  PRC_SendeKanalOeffnen()
  IF N_PRC_Err1 <> N_PRC_MsgOff THEN
    RETURN(N_PRC_Err1)
  ENDIF
  O_PRC_Data2 = 0
  O_PRC_Data1 = N_PRC_ID
  IF NOT PRC_DatenSenden() THEN
    RETURN(N_PRC_Err1)
  ENDIF
  PRC_SendeKanalSchliessen()
  IF NOT PRC_DatenEmpfangen() THEN
    RETURN(N_PRC_Err1)
  ENDIF
  PRC_EmpfKanalSchliessen()               ; PRC_EmpfKanalSchliessen
  PRC_EmpfDatenAuswerten()                ; PRC_EmpfDatenAuswerten
  IF N_PRC_IDAck <> N_PRC_ID THEN
    N_PRC_Err1   = N_PRC_MsgOff + 43      ; falsche RETURNID
    B_PRC_MsgFlg = TRUE
    RETURN(N_PRC_Err1)
  ENDIF
  SWITCH N_PRC_KennAck
    CASE 0
      N_PRC_Err1   = N_PRC_MsgOff         ; Perceptron bereit
    CASE 5
      N_PRC_Err1   = N_PRC_MsgOff + 7     ; Perceptron von diesem Roboter bereits gestartet
    CASE 12
      N_PRC_Err1   = N_PRC_MsgOff + 6     ; Perceptron offline
    CASE 23
      N_PRC_Err1   = N_PRC_MsgOff + 23    ; Kalibriermodus
    CASE 24
      N_PRC_Err1   = N_PRC_MsgOff + 24    ; Teachmodus
    CASE 29
      N_PRC_Err1   = N_PRC_MsgOff + 29    ; BaseFinder
    CASE 30
      N_PRC_Err1   = N_PRC_MsgOff + 30    ; ToolFinder
    CASE 255
      N_PRC_Err1   = N_PRC_MsgOff + 8     ; allg. Fehler
    DEFAULT
      N_PRC_Err1   = N_PRC_MsgOff + 9     ; Fehler nicht spezifiziert
  ENDSWITCH
  RETURN(N_PRC_Err1)
ENDFCT
;
  ;ENDFOLD (Get Status)
;
  ;FOLD Punkt Messung
;
DEF PRC_PunktMessung(nPktNr:IN,nFrame:IN,nTool:IN)
INT nPktNr
INT nFrame
INT nTool
INT nMPTimerStart
INT nComTimerStart
  N_PRC_Err1   = 200
  B_PRC_MsgFlg = FALSE
  IF (NOT I_PRC_Zyklus) AND (NOT I_PRC_PgmMod) THEN
    B_PRC_MsgFlg = TRUE
    N_PRC_Err1   = 224   ; Messung nicht gestartet
    RETURN
  ENDIF
  O_PRC_PktNr = nPktNr
  O_PRC_Pkt   = TRUE
  nMPTimerStart = $Rob_Timer
  wait for (I_PRC_PktAck OR I_PRC_PosInf OR ((($Rob_Timer - nMPTimerStart) > N_PRC_TmMP) AND NOT I_PRC_PgmMod))
  IF (($Rob_Timer - nMPTimerStart) > N_PRC_TmMP) AND NOT I_PRC_PgmMod THEN
    N_PRC_Err1   = 225   ; Timeout beim warten auf Messungende
    B_PRC_MsgFlg = TRUE
    O_PRC_PktNr  = 0
    O_PRC_Pkt    = FALSE
    RETURN
  ENDIF
  IF I_PRC_Fehler THEN   ; Perceptron Fehler bei PRC_PunktMessung
    B_PRC_MsgFlg = TRUE
    SWITCH I_PRC_FehlNr
      CASE 1
        N_PRC_Err1 = 223   ; PositionsID ungueltig
      CASE 5
        N_PRC_Err1 = 224   ; Messytstem nicht gestartet
      CASE 18
        N_PRC_Err1 = 213   ; Allgemeiner Fehler
      CASE 19
        N_PRC_Err1 = 227   ; Falsche Punktreihenfolge
CASE 512
        N_PRC_Err1 = 213   ; Allgemeiner Fehler
        IF B_PRC_ISTOOL == TRUE THEN
          N_PRC_Err1   = 228   ; Nur im ToolFinder-Modus (Messfehler)
          B_PRC_MsgFlg = FALSE
        ENDIF
        IF B_PRC_ISBASE == TRUE THEN
          N_PRC_Err1   = 229   ; Nur im BaseFinder-Modus (Messfehler)
          B_PRC_MsgFlg = FALSE
        ENDIF
      DEFAULT
    ENDSWITCH
    O_PRC_PktNr = 0
    O_PRC_Pkt   = FALSE
    RETURN
  ENDIF
  IF I_PRC_PosInf THEN
	IF (nFrame == -1) OR (nTool == -1) THEN
	  PRC_SendInfo (3,N_PRC_CurMod,nPktNr) ; Sende Poseinfo (3)
	ELSE
     N_PRC_BasNr = $ACT_BASE
     N_PRC_TooNr = $ACT_TOOL
	  PRC_SendInfo (13,N_PRC_CurMod,nPktNr,N_PRC_BasNr,N_PRC_TooNr) ; Sende Pose ID (13)
	ENDIF
	IF (N_PRC_Err1 <> N_PRC_MsgOff) AND (B_PRC_MsgFlg) THEN
      N_PRC_Ret1 = PRC_MsgErr(#NotifyMsg,N_PRC_Err1)
    ENDIF
  ENDIF
  nMPTimerStart = $Rob_Timer
  wait for (I_PRC_PktAck OR ((($Rob_Timer - nMPTimerStart) > N_PRC_TmMP) AND NOT I_PRC_PgmMod))
  O_PRC_Pkt   = FALSE
  O_PRC_PktNr = 0
  IF (($Rob_Timer - nMPTimerStart) > N_PRC_TmMP) AND NOT I_PRC_PgmMod THEN
    N_PRC_Err1   = 225   ; Timeout beim warten auf Messungende
    B_PRC_MsgFlg = TRUE
    RETURN
  ENDIF
  nComTimerStart = $Rob_Timer
  wait for (NOT(I_PRC_PktAck) OR ((($Rob_Timer - nComTimerStart) > N_PRC_TmCom) AND NOT I_PRC_PgmMod))
  IF (($Rob_Timer - nComTimerStart) > N_PRC_TmCom) AND NOT I_PRC_PgmMod THEN
    N_PRC_Err1   = 225   ; Timeout beim warten auf Messungende
    B_PRC_MsgFlg = TRUE
    RETURN
  ENDIF
END
;
  ;ENDFOLD (Punkt Messung)
;
  ;FOLD Start Scan
;
DEF PRC_StartScan(nScanSct:IN)
INT nScanSct
INT nMPTimerStart
INT nScanTimerStart
  IF (NOT I_PRC_Zyklus) AND (NOT I_PRC_PgmMod) THEN
    B_PRC_MsgFlg = TRUE
    N_PRC_ERR1   = 284     ; Messung nicht gestartet
    RETURN
  ENDIF
  IF I_PRC_SScAck THEN
    B_PRC_MsgFlg = TRUE
    N_PRC_ERR1   = 291     ; StartScanAck nicht zurueckgenommen
    RETURN
  ENDIF
  nScanTimerStart = $Rob_Timer
  O_PRC_PktNr     = nScanSct
  O_PRC_SSc       = TRUE
  nMPTimerStart   = $Rob_Timer
  wait for (I_PRC_SScAck OR I_PRC_PosInf OR ((($Rob_Timer - nMPTimerStart) > N_PRC_TmMP) AND NOT I_PRC_PgmMod))
  IF (($Rob_Timer - nMPTimerStart) > N_PRC_TmMP) THEN
    N_PRC_Err1   = 292       ; StartScanAck nicht gesetzt
    B_PRC_MsgFlg = TRUE
    O_PRC_PktNr  = 0
    O_PRC_SSc    = FALSE
    RETURN
  ENDIF
  IF I_PRC_Fehler THEN       ;Perceptron Fehler bei PRC_PunktMessung
    SWITCH I_PRC_FehlNr
      CASE 1
        N_PRC_Err1   = 283   ; PositionsID ungueltig
        B_PRC_MsgFlg = TRUE
      CASE 5
        N_PRC_Err1   = 284   ; Messytstem nicht gestartet
        B_PRC_MsgFlg = TRUE
      CASE 18
        N_PRC_Err1   = 285   ; Allgemeiner Fehler
        B_PRC_MsgFlg = TRUE
      DEFAULT
    ENDSWITCH
    O_PRC_PktNr = 0
    O_PRC_SSc   = FALSE
    RETURN
  ENDIF
  IF I_PRC_PosInf THEN
	PRC_SendInfo(3,N_PRC_CurMod,nScanSct) ; Sende Poseinfo (3)
    IF (N_PRC_Err1 <> N_PRC_MsgOff) AND (B_PRC_MsgFlg) THEN
      N_PRC_Ret1 = PRC_MsgErr(#NotifyMsg,N_PRC_Err1)
    ENDIF
    nMPTimerStart = $Rob_Timer
    wait for (I_PRC_SScAck OR (($Rob_Timer - nMPTimerStart) > N_PRC_TmMP))
    IF (($Rob_Timer - nMPTimerStart) > N_PRC_TmMP) THEN
      N_PRC_Err1   = 292   ; StartScanAck nicht gesetzt
      B_PRC_MsgFlg = TRUE
      O_PRC_PktNr  = 0
      O_PRC_SSc    = FALSE
      RETURN
    ENDIF
  ENDIF
  O_PRC_SSc    = FALSE
  O_PRC_StrVrz = $Rob_Timer - nScanTimerStart
END
;
  ;ENDFOLD (Start Scan)
;
  ;FOLD End Scan
;
DEFFCT INT PRC_EndScan(nScanSct:IN)
REAL rVelocity
INT  nScanSct
INT  nErr
INT  nByte01
INT  nByte02
INT  nByte03
INT  nByte04
INT  nMPTimerStart
INT  nScanTimerStart
  IF (NOT I_PRC_Zyklus) AND (NOT I_PRC_PgmMod) THEN
    B_PRC_MsgFlg = TRUE
    RETURN(284)  ; Messung nicht gestartet
  ENDIF
  IF I_PRC_EScAck THEN
    B_PRC_MsgFlg = TRUE
    RETURN(281)  ; EndScanAck nicht zurueckgenommen
  ENDIF
  nScanTimerStart = $Rob_Timer
  O_PRC_PktNr     = nScanSct
  rVelocity       = $VEL.CP * ($OV_ROB / 100.0) * 1000
  PRC_ConvReal2Bytes(rVelocity,nByte01,nByte02,nByte03,nByte04 )
  O_PRC_Speed1    = nByte01
  O_PRC_Speed2    = nByte02
  O_PRC_Speed3    = nByte03
  O_PRC_Speed4    = nByte04
  O_PRC_ESc       = TRUE
  nMPTimerStart = $Rob_Timer
  WAIT FOR (I_PRC_EScAck OR I_PRC_PosInf OR ((($Rob_Timer - nMPTimerStart) > N_PRC_TmMP) AND NOT I_PRC_PgmMod))
  IF (($Rob_Timer - nMPTimerStart) > N_PRC_TmMP) THEN
    O_PRC_PktNr  = 0
    O_PRC_ESc    = FALSE
    O_PRC_Speed1 = 0
    O_PRC_Speed2 = 0
    O_PRC_Speed3 = 0
    O_PRC_Speed4 = 0
    B_PRC_MsgFlg = TRUE
    RETURN(282)  ; EndScanAck nicht gesetzt
  ENDIF
  IF I_PRC_Fehler THEN   ; Perceptron Fehler bei PRC_EndScan
    B_PRC_MsgFlg = TRUE
    SWITCH I_PRC_FehlNr
      CASE 1
        nErr = 283  ; PositionsID ungueltig
      CASE 5
        nErr = 284  ; Messytstem nicht gestartet
      CASE 18
        nErr = 285  ; Allgemeiner Fehler
      DEFAULT
        nErr = 286  ; Fehler nicht spezifiziert
    ENDSWITCH
    O_PRC_PktNr  = 0
    O_PRC_Speed1 = 0
    O_PRC_Speed2 = 0
    O_PRC_Speed3 = 0
    O_PRC_Speed4 = 0
    O_PRC_ESc    = FALSE
    RETURN(nErr)
  ENDIF
  IF I_PRC_PosInf THEN
	PRC_SendInfo(3,N_PRC_CurMod,nScanSct) ; Sende Poseinfo (3)
	IF (N_PRC_Err1 <> N_PRC_MsgOff) AND (B_PRC_MsgFlg) THEN
      N_PRC_Ret1 = PRC_MsgErr(#NotifyMsg,N_PRC_Err1)
    ENDIF
    nMPTimerStart = $Rob_Timer
    WAIT FOR (I_PRC_EScAck OR (($Rob_Timer - nMPTimerStart) > N_PRC_TmMP))
    IF (($Rob_Timer - nMPTimerStart) > N_PRC_TmMP) THEN
      O_PRC_PktNr = 0
      O_PRC_ESc   = FALSE
      B_PRC_MsgFlg = TRUE
      RETURN(282)   ; EndScanAck nicht gesetzt
    ENDIF
  ENDIF
  O_PRC_PktNr   = 0
  O_PRC_EndVrz  = $Rob_Timer - nScanTimerStart
  O_PRC_ESc     = FALSE
  nMPTimerStart = $Rob_Timer
  WAIT FOR (I_PRC_EScAck OR (($Rob_Timer - nMPTimerStart) > N_PRC_TmMP))
  IF (($Rob_Timer - nMPTimerStart) > N_PRC_TmMP) THEN
    B_PRC_MsgFlg = TRUE
    RETURN(282)   ; EndScanAck nicht gesetzt
  ENDIF
  RETURN(0)
ENDFCT
;
  ;ENDFOLD (End Scan)
;
  ;FOLD Set Korr
;
DEF PRC_SetKorrektur (VFNR:IN)
INT VFNR
  IF (B_PRC_VFErr == TRUE) THEN
    IF $ACT_BASE == 0 THEN
      BASE_DATA[N_PRC_KorBas] = $Nullframe
    ELSE
      BASE_DATA[N_PRC_KorBas] = BASE_DATA[$ACT_BASE]
    ENDIF
    N_PRC_Err1         = 1046
    $FLAG[F_PRC_VFErr] = TRUE
    $FLAG[F_PRC_Err]   = TRUE
    $FLAG[F_PRC_NoErr] = FALSE
  ELSE
    IF $ACT_BASE == 0 THEN
      BASE_DATA[N_PRC_KorBas] = AVF_PRC_Korr[VFNR]
    ELSE
      BASE_DATA[N_PRC_KorBas] = BASE_DATA[$ACT_BASE] : AVF_PRC_Korr[VFNR]
    ENDIF
    $FLAG[F_PRC_VFErr] = FALSE
    $FLAG[F_PRC_Err]   = FALSE
    $FLAG[F_PRC_NoErr] = TRUE
    N_PRC_Err1         = 1000
  ENDIF
END
;
  ;ENDFOLD (Set Korr)
;
  ;FOLD Get Korr
;
DEF PRC_GetKorrektur (TYP:IN,SUBTYP:IN,VFNR:IN,PAR2:IN)
INT TYP
INT SUBTYP
INT VFNR
INT PAR2
INT nByte1
INT nByte2
  B_PRC_MsgFlg = FALSE
  AVF_PRC_Korr[VFNR] = $NULLFRAME
  ; Korrektur abholen
  PRC_SendeKanalOeffnen()
  IF N_PRC_Err1 <> N_PRC_MsgOff THEN
    GOTO Get_Korr_Err
  ENDIF
  O_PRC_Data2 = 0 ; leer
  O_PRC_Data1 = 6 ; ID
  PRC_ConvWort2Byte(VFNR,nByte2,nByte1)
  O_PRC_Data3 = nByte1
  O_PRC_Data4 = nByte2
  PRC_ConvWort2Byte(3,nByte2,nByte1)
  O_PRC_Data5 = nByte1
  O_PRC_Data6 = nByte2
  IF NOT PRC_DatenSenden() THEN
    GOTO Get_Korr_Err
  ENDIF
  PRC_SendeKanalSchliessen()
  IF NOT PRC_DatenEmpfangen() THEN
    GOTO Get_Korr_Err
  ENDIF
  PRC_EmpfKanalSchliessen()
  PRC_EmpfDatenAuswerten()
  IF N_PRC_IDAck <> 6 THEN
    N_PRC_Err1   = 1043 ;falsche RETURNID
    GOTO Get_Korr_Err
  ENDIF
  IF N_PRC_P1Ack <> VFNR THEN
    N_PRC_Err1   = 1038 ;Falsche RETURN Fixnr
    GOTO Get_Korr_Err
  ENDIF
  IF N_PRC_P2Ack <> 0 THEN
    N_PRC_Err1   = 1042 ;keine Korrekturwerte vorhanden
    GOTO Get_Korr_Err
  ENDIF
  GOTO Get_Korr_OK
Get_Korr_Err:
  B_PRC_VFErr = TRUE
  $FLAG[F_PRC_VFErr]  = TRUE
  $FLAG[F_PRC_Err]    = TRUE
  $FLAG[F_PRC_NoErr]  = FALSE
  AVF_PRC_Korr[VFNR] = $Nullframe
  VF_PRC_Sen          = $Nullframe
  RETURN
Get_Korr_OK:
  B_PRC_VFErr = FALSE
  IF PRC_CheckMaxVF(VF_PRC_Sen) THEN
    AVF_PRC_Korr[VFNR] = VF_PRC_Sen
    N_PRC_Err1          = 1000
  ELSE
    B_PRC_VFErr = TRUE
    $FLAG[F_PRC_VFMax] = TRUE
    $FLAG[F_PRC_VFErr] = TRUE
    $FLAG[F_PRC_Err]   = TRUE
    $FLAG[F_PRC_NoErr] = FALSE
    AVF_PRC_Korr[VFNR] = $Nullframe
    VF_PRC_Sen          = $Nullframe
  ENDIF
END
;
  ;ENDFOLD (Get Korr)
;
  ;FOLD Start Messung
;
DEF PRC_StartMessung(TYP:IN,SUBTYP:IN,PAR2:IN)
INT TYP
INT SUBTYP
INT PAR2
INT nByte1
INT nByte2
  N_PRC_ID     = 1
  B_PRC_StrSPS = FALSE
  PRC_SendeKanalOeffnen()
  IF N_PRC_Err1 <> N_PRC_MsgOff THEN
    RETURN
  ENDIF
  O_PRC_Data2 = 0                         ;JSN,AuxID,ColorCode,AuxID-String
  O_PRC_Data1 = N_PRC_ID                  ;ID
  PRC_ConvWort2Byte(TYP,nByte2,nByte1)    ;Modell HL Byte gedreht!!!
  O_PRC_Data3 = nByte1
  O_PRC_Data4 = nByte2
  PRC_ConvWort2Byte(SUBTYP,nByte2,nByte1) ;Routine HL Byte gedreht!!!
  O_PRC_Data5 = nByte1
  O_PRC_Data6 = nByte2
  IF NOT PRC_DatenSenden() THEN
    RETURN
  ENDIF
  PRC_SendeKanalSchliessen()
  IF NOT PRC_DatenEmpfangen() THEN
    RETURN
  ENDIF
  PRC_EmpfKanalSchliessen()
  PRC_EmpfDatenAuswerten()
  SWITCH N_PRC_KennAck
    CASE 0
      N_PRC_Err1   = N_PRC_MsgOff      ; Befehl ok
    CASE 1
      N_PRC_Err1   = N_PRC_MsgOff + 5  ; Modell od. Routine nicht definiert
    CASE 5
      N_PRC_Err1   = N_PRC_MsgOff + 7  ; Perceptron bereits gestartet
    CASE 12
      N_PRC_Err1   = N_PRC_MsgOff + 6  ; Perceptron offline
    CASE 254
      N_PRC_Err1   = N_PRC_MsgOff + 12 ; Perceptron von SPS gestartet
    CASE 255
      N_PRC_Err1   = N_PRC_MsgOff + 8  ; allg. Fehler
    DEFAULT
      N_PRC_Err1   = N_PRC_MsgOff + 9  ; Fehler nicht spezifiziert
  ENDSWITCH
  IF N_PRC_Err1 <> N_PRC_MsgOff THEN
    IF N_PRC_Err1 == (N_PRC_MsgOff + 7) THEN
      PRC_DebugDlg(11,0,0)
      B_PRC_StrSPS = TRUE
    ENDIF
    RETURN
  ENDIF
  IF N_PRC_IDAck <> N_PRC_ID THEN
    N_PRC_Err1    = N_PRC_MsgOff + 43  ;falsche RETURNID
  ELSE
    IF (N_PRC_P1Ack <> TYP) THEN
      N_PRC_Err1   = N_PRC_MsgOff + 11 ;falsche RETURN ModellNr
    ENDIF
  ENDIF
END
;
  ;ENDFOLD (Start Messung)
;
  ;FOLD Start UP Messung
;
DEF PRC_StartUpMess (TYP:IN,SUBTYP:IN,PAR2:IN)
INT TYP
INT SUBTYP
INT PAR2
INT nByte1
INT nByte2
  ;holt nur UP-Nr von Perceptron wenn Perc von SPS gestartet
  N_PRC_ID = 11
  PRC_SendeKanalOeffnen()
  IF N_PRC_Err1 <> N_PRC_MsgOff THEN
    RETURN
  ENDIF
  O_PRC_Data2 = 0        ;JSN,AuxID,ColorCode,AuxID-String
  O_PRC_Data1 = N_PRC_ID ;ID
  PRC_ConvWort2Byte(TYP,nByte2,nByte1)
  O_PRC_Data3 = nByte1
  O_PRC_Data4 = nByte2
  PRC_ConvWort2Byte(SUBTYP,nByte2,nByte1)
  O_PRC_Data5 = nByte1
  O_PRC_Data6 = nByte2
  IF NOT PRC_DatenSenden() THEN
    RETURN
  ENDIF
  PRC_SendeKanalSchliessen()
  IF NOT PRC_DatenEmpfangen() THEN
    RETURN
  ENDIF
  PRC_EmpfKanalSchliessen()
  PRC_EmpfDatenAuswerten()
  SWITCH N_PRC_KennAck
    CASE 0
      N_PRC_Err1 = N_PRC_MsgOff      ; Befehl ok
    CASE 1
      N_PRC_Err1 = N_PRC_MsgOff + 5  ; Modell od. Routine nicht definiert
    CASE 5
      N_PRC_Err1 = N_PRC_MsgOff + 7  ; Perceptron von SPS nicht gestartet
    CASE 12
      N_PRC_Err1 = N_PRC_MsgOff + 6  ; Perceptron offline
    CASE 255
      N_PRC_Err1 = N_PRC_MsgOff + 8  ; allg. Fehler
    DEFAULT
      N_PRC_Err1 = N_PRC_MsgOff + 9  ; Fehler nicht spezifiziert
  ENDSWITCH
  IF N_PRC_Err1 <> N_PRC_MsgOff THEN
    RETURN
  ENDIF
  IF N_PRC_IDAck <> N_PRC_ID THEN
    N_PRC_Err1 = N_PRC_MsgOff + 43   ; Falsche RETURNID
  ELSE
    IF N_PRC_P1Ack <> TYP THEN
      N_PRC_Err1 = N_PRC_MsgOff + 11 ; Falsche RETURN ModellNr
    ENDIF
  ENDIF
END
;
;ENDFOLD (Start UP Messung)
;
;FOLD Start UP Komp
;
DEF PRC_StartUpKomp (TYP:IN,SUBTYP:IN,PAR2:IN)
INT TYP
INT SUBTYP
INT PAR2
INT nByte1
INT nByte2
  N_PRC_ID = 12
  PRC_SendeKanalOeffnen()
  IF N_PRC_Err1 <> N_PRC_MsgOff THEN
    RETURN
  ENDIF
  O_PRC_Data2 = 0        ; JSN,AuxID,ColorCode,AuxID-String
  O_PRC_Data1 = N_PRC_ID ; ID
  PRC_ConvWort2Byte(TYP,nByte2,nByte1)
  O_PRC_Data3 = nByte1
  O_PRC_Data4 = nByte2
  PRC_ConvWort2Byte(SUBTYP,nByte2,nByte1)
  O_PRC_Data5 = nByte1
  O_PRC_Data6 = nByte2
  IF NOT PRC_DatenSenden() THEN
    RETURN
  ENDIF
  PRC_SendeKanalSchliessen()
  IF NOT PRC_DatenEmpfangen() THEN
    RETURN
  ENDIF
  PRC_EmpfKanalSchliessen()
  PRC_EmpfDatenAuswerten()
  SWITCH N_PRC_KennAck
    CASE 0
      N_PRC_Err1 = N_PRC_MsgOff + 50 ; Kompensation ok (nicht erforderlich)
    CASE 1
      N_PRC_Err1 = N_PRC_MsgOff + 51 ; Kompensation erforderlich (Voll)
    CASE 2
      N_PRC_Err1 = N_PRC_MsgOff + 52 ; Kompensation erforderlich (Split)
    CASE 4
      N_PRC_Err1 = N_PRC_MsgOff + 53 ; Kompensation deaktiviert (SPS)
    CASE 6
      N_PRC_Err1 = N_PRC_MsgOff + 54 ; Modell/UP ungueltig
    CASE 16
      N_PRC_Err1 = N_PRC_MsgOff + 60 ; Perceptron im falschen Status
    CASE 32
      N_PRC_Err1 = N_PRC_MsgOff + 61 ; Perceptron in der Startprozedur
    CASE 64
      N_PRC_Err1 = N_PRC_MsgOff + 70 ; Fehler in der Startprozedur
    CASE 128
      N_PRC_Err1 = N_PRC_MsgOff + 71 ; Fehler in der Kompensation (Konfiguration)
    DEFAULT
      N_PRC_Err1 = N_PRC_MsgOff + 9  ; Fehler nicht spezifiziert
  ENDSWITCH
  IF N_PRC_Err1 <> N_PRC_MsgOff THEN
    RETURN
  ENDIF
  IF N_PRC_IDAck <> N_PRC_ID THEN
    N_PRC_Err1 = N_PRC_MsgOff + 43   ; Falsche RETURNID
  ELSE
    IF N_PRC_P1Ack <> TYP THEN
      N_PRC_Err1 = N_PRC_MsgOff + 11 ; Falsche RETURN ModellNr
    ENDIF
  ENDIF
END
;
  ;ENDFOLD (Start UP Komp)
;
  ;FOLD Reset
;
DEFFCT INT PRC_Reset()
INT nComTimerStart
  O_PRC_Reset = TRUE
  nComTimerStart = $Rob_Timer
  WAIT FOR (I_PRC_Reset OR (($Rob_Timer - nComTimerStart) > N_PRC_TmCom))
  O_PRC_Reset = FALSE
  IF (($Rob_Timer - nComTimerStart) > N_PRC_TmCom) THEN
    RETURN(521)  ; Timeout bei Reset Perceptron
  ELSE
    nComTimerStart = $Rob_Timer
    WAIT FOR (NOT(I_PRC_Reset) OR (($Rob_Timer - nComTimerStart) > N_PRC_TmCom))
    IF (($Rob_Timer - nComTimerStart) > N_PRC_TmCom) THEN
      RETURN(522)  ; Timeout bei Reset Perceptron
    ENDIF
  ENDIF
  RETURN (0)
ENDFCT
;
  ;ENDFOLD (Reset)
;
  ;FOLD Messung Beenden
;
DEF PRC_MessungBeenden(CMD_SEL:IN)
INT CMD_SEL
INT nComTimerStart
  O_PRC_ME = TRUE   ; End Measurement
  nComTimerStart = $Rob_Timer
  wait for (I_PRC_MEACK OR (($Rob_Timer - nComTimerStart) > N_PRC_TmCom))
  IF (($Rob_Timer - nComTimerStart) > N_PRC_TmCom) THEN   ;timeout beim warten auf I_PRC_MEACK
    N_PRC_Err1   = N_PRC_MsgOff + 4
    B_PRC_MsgFlg = TRUE
    RETURN
  ENDIF
  O_PRC_ME = FALSE
  IF NOT PRC_EmpfangsKanalOeffnen() THEN
    B_PRC_MsgFlg = TRUE
    RETURN
  ENDIF
  IF NOT PRC_DatenEmpfangen() THEN
    B_PRC_MsgFlg = TRUE
    RETURN
  ENDIF
  PRC_EmpfKanalSchliessen()
  nComTimerStart = $Rob_Timer
  wait for (NOT I_PRC_MEACK OR (($Rob_Timer - nComTimerStart) > N_PRC_TmCom))
  PRC_EmpfDatenAuswerten()
  IF N_PRC_IDAck <> 7 THEN ;Falsche Antwort auf MessEnde
    N_PRC_Err1   = N_PRC_MsgOff + 43
    B_PRC_MsgFlg = TRUE
    RETURN
  ENDIF
  SWITCH CMD_SEL
    CASE 1001                 ; IMT  ; Hauptgruppe 9, Untergruppe 1
      SWITCH N_PRC_KennAck
        CASE 0,1 ; Messung Ende
        CASE 4
          N_PRC_Err1   = N_PRC_MsgOff + 24         ; Messung ist nicht gestartet
          B_PRC_MsgFlg = TRUE
          RETURN
        DEFAULT
          N_PRC_Err1   = N_PRC_MsgOff + 43         ; Parameter-Kennung nicht definiert
          B_PRC_MsgFlg = TRUE
          RETURN
      ENDSWITCH
      SWITCH N_PRC_P1Ack
        CASE 0                              ; alles ok
          N_PRC_Err1   = N_PRC_MsgOff
        CASE 1
          N_PRC_Err1   = 1151   ; Robot 1 SensorError
          ;N_PRC_Err1 = N_PRC_MsgOff + 1  ; Trend bei Messende
        CASE 2
          N_PRC_Err1   = 1152   ; Robot 1 SensorToleranz
          ;N_PRC_Err1 = N_PRC_MsgOff + 2  ; Spec bei Messende
        CASE 3
          N_PRC_Err1 = N_PRC_MsgOff + 3  ; Trend+Spec bei Messende
        CASE 4
          N_PRC_Err1   = 1153   ; Robot 1 VF Error
          ;N_PRC_Err1 = N_PRC_MsgOff + 4  ; Reject bei Messende
        CASE 5
          N_PRC_Err1 = N_PRC_MsgOff + 5  ; Reject+Trend bei Messende
        CASE 6
          N_PRC_Err1 = N_PRC_MsgOff + 6  ; Reject+Spec bei Messende
        CASE 7
          N_PRC_Err1 = N_PRC_MsgOff + 7  ; Reject+Trend+Spec bei Messende
        CASE 8,9,10,11,12,13,14,15
          N_PRC_Err1   = 1154   ; Robot 1 VF Toleranz
          ;N_PRC_Err1 = N_PRC_MsgOff + 8   ; Error bei Messende
        CASE 16
          N_PRC_Err1   = 1155   ; Robot 2 SensorError
        CASE 32
          N_PRC_Err1   = 1156   ; Robot 2 SensorToleranz
        CASE 48
          N_PRC_Err1 = N_PRC_MsgOff + 3  ; Robot 2 Trend+Spec bei Messende
        CASE 64
          N_PRC_Err1   = 1157   ; Robot 2 VF Error
        CASE 80
          N_PRC_Err1 = N_PRC_MsgOff + 5  ; Robot 2 Reject+Trend bei Messende
        CASE 96
          N_PRC_Err1 = N_PRC_MsgOff + 6  ; Robot 2 Reject+Spec bei Messende
        CASE 112
           N_PRC_Err1 = N_PRC_MsgOff + 7  ; Robot 2 Reject+Trend+Spec bei Messende
        CASE 128, 144, 160, 176, 192, 208, 224, 240
          N_PRC_Err1   = 1158   ; Robot 2 VF Toleranz
        DEFAULT
          N_PRC_Err1   = N_PRC_MsgOff + 36         ; Ungueltiger Par1 bei Messende
          B_PRC_MsgFlg = TRUE
      ENDSWITCH
    CASE 1002 ; AutoGuide  ; Hauptgruppe 9, Untergruppe 2
      SWITCH N_PRC_KennAck
        CASE 0 ; Messung Ende
        CASE 4
          N_PRC_Err1   = N_PRC_MsgOff + 24         ; Messung ist nicht gestartet
          B_PRC_MsgFlg = TRUE
          RETURN
        DEFAULT
          N_PRC_Err1   = N_PRC_MsgOff + 43         ; Parameter-Kennung nicht definiert
          B_PRC_MsgFlg = TRUE
          RETURN
      ENDSWITCH
      SWITCH N_PRC_P1Ack
        CASE 0                              ; alles ok
          N_PRC_Err1   = N_PRC_MsgOff
        CASE 1
          N_PRC_Err1   = 1151   ; Robot 1 SensorError
        CASE 2
          N_PRC_Err1   = 1152   ; Robot 1 SensorToleranz
        CASE 4
          N_PRC_Err1   = 1153   ; Robot 1 VF Error
        CASE 8
          N_PRC_Err1   = 1154   ; Robot 1 VF Toleranz
        CASE 16
          N_PRC_Err1   = 1155   ; Robot 2 SensorError
        CASE 32
          N_PRC_Err1   = 1156   ; Robot 2 SensorToleranz
        CASE 64
          N_PRC_Err1   = 1157   ; Robot 2 VF Error
        CASE 128
          N_PRC_Err1   = 1158   ; Robot 2 VF Toleranz
        DEFAULT
          IF N_PRC_P1Ack < 16 THEN
            N_PRC_Err1   = 1159  ; Rob 1 mehrere Fehler
            B_PRC_MsgFlg = TRUE
          ELSE
            IF N_PRC_P1Ack < 256 THEN
              N_PRC_Err1   = 1160  ; Rob 2 mehrere Fehler
              B_PRC_MsgFlg = TRUE
            ELSE
              N_PRC_Err1   = N_PRC_MsgOff + 36 ; Ungueltiger Par1 bei Messende
              B_PRC_MsgFlg = TRUE
            ENDIF
          ENDIF
      ENDSWITCH
    CASE 1003                 ; AutoGauge  ; Hauptgruppe 9, Untergruppe 3
  ENDSWITCH
END
;
  ;ENDFOLD (Messung Beenden)
;
  ;FOLD Sys-Init-1
;
DEF PRC_SysInit1(nSUBSYSTEM:IN,nCONVEYORTECH:IN,nUSELIFEBIT:IN,nFRAME:IN,nVF:IN,nRESERVE:IN) ; System Einstellungen 1
INT nSUBSYSTEM ;    Toolkalibrier-Modus = 0-ToolFinder/1=Temperaturkalibrierung
INT nCONVEYORTECH ; 0=Ohne/1=Mit
INT nUSELIFEBIT ;   0=Ohne/1=Mit
INT nFRAME ;        KorrekturBase (Default 31, Conveyor 11)
INT nVF ;           VFNr fuer Robotertausch
INT nRESERVE ;      Frei
  ; Alle Variabeln auf Default
  PRC_DefaultInit()
  SWITCH nSUBSYSTEM
    CASE 0 ; Toolkalibrier-Modus = ToolFinder
	  N_PRC_SubSystem = 0
	CASE 1 ; Toolkalibrier-Modus = Temperaturkalibrierung
	  N_PRC_SubSystem = 1
	DEFAULT ; ncht definiert
	  B_PRC_MsgKri = TRUE
	  N_PRC_Ret1   = PRC_MsgErr(#NotifyMsg,1200,nSUBSYSTEM)
  ENDSWITCH
  SWITCH nCONVEYORTECH
    CASE 0 ; Ohne
	  B_PRC_CoTech = FALSE
     IF (nFRAME >= 1) AND (nFRAME <= 31) THEN
       N_PRC_KorBas = nFRAME
     ELSE
       N_PRC_KorBas = 31
       B_PRC_MsgKri = TRUE
	    N_PRC_Ret1   = PRC_MsgErr(#NotifyMsg,1202,nFRAME)
     ENDIF
	CASE 1 ; Mit
	  B_PRC_CoTech  = TRUE
     N_PRC_KorBas  = 11
	DEFAULT ; ncht definiert
	  B_PRC_MsgKri = TRUE
	  N_PRC_Ret1   = PRC_MsgErr(#NotifyMsg,1201,nCONVEYORTECH)
  ENDSWITCH
  IF nUSELIFEBIT == 0 THEN
     B_PRC_UseFct = FALSE
  ELSE
     B_PRC_UseFct = TRUE
  ENDIF
  N_PRC_VFNr = nVF
END
;
  ;ENDFOLD (Sys-Init-1)
;
  ;FOLD Sys-Init-2
;
DEF PRC_SysInit2(nTIMEOUTMP:IN,nTIMEOUTCOM:IN,nERRFLAGS:IN,nSIGNALS:IN,nINTERRUPT1:IN,nINTERRUPT2:IN) ; System Einstellungen 2
INT nTIMEOUTMP ;   Timeout Messpunkt     [ms]
INT nTIMEOUTCOM ;  Timeout Kommunikation [ms]
INT nERRFLAGS ;    Start Fehler-Flags
INT nSIGNALS ;     Start Master-Signale
INT nINTERRUPT1 ;  Interrupt fuer RobMove
INT nINTERRUPT2 ;  Interrupt fuer RobNoMove
   ; Timeout Messpunkt     [ms]
   N_PRC_TmMP  = nTIMEOUTMP
   ; Timeout Kommunikation [ms]
   N_PRC_TmCom = nTIMEOUTCOM
   ; Fehler-Flags
   N_PRC_FiErr = nERRFLAGS      ; Erstes Fehler Flag
   F_PRC_NoErr = nERRFLAGS      ; Kein Fehler
   F_PRC_Err   = nERRFLAGS + 1  ; Fehler
   F_PRC_GeStr = nERRFLAGS + 2  ; Sammel Stoerung
   F_PRC_TmOut = nERRFLAGS + 3  ; TimeOut
   F_PRC_NoVal = nERRFLAGS + 4  ; Kein Auftrag
   F_PRC_SyIna = nERRFLAGS + 5  ; System Inaktiv
   F_PRC_SyAkt = nERRFLAGS + 6  ; System Aktiv
   F_PRC_NoStr = nERRFLAGS + 7  ; Kein Messstart von SPS
   F_PRC_ModID = nERRFLAGS + 8  ; Falsche Modell ID
   F_PRC_VFMax = nERRFLAGS + 9  ; Maximale Korrekturwerte erreicht
   F_PRC_VFErr = nERRFLAGS + 10 ; Korrekturwerte nicht vorhanden
   ; Master-Signale
   N_PRC_MaSig = nSIGNALS
   N_PRC_SigLB = nSIGNALS
   ;Interrupt fuer RobMove
   N_PRC_Int1 = nINTERRUPT1
   ;Interrupt fuer RobNoMove
   N_PRC_Int2 = nINTERRUPT2
END
;
  ;ENDFOLD (Sys-Init-2)
;
  ;FOLD Model-Init
;
DEF PRC_ModelInit(nMODEL1:IN,nMODEL2:IN,nMODEL3:IN,nMODEL4:IN,nMODEL5:IN,nMODEL6:IN) ; ModelInit (Mehrfach Aufruf erlaubt)
INT nMODEL1 ; Freigegebenes Modell 1
INT nMODEL2 ; Freigegebenes Modell 2
INT nMODEL3 ; Freigegebenes Modell 3
INT nMODEL4 ; Freigegebenes Modell 4
INT nMODEL5 ; Freigegebenes Modell 5
INT nMODEL6 ; Freigegebenes Modell 6
INT nCounterModels
INT nTyp
  FOR nCounterModels = 1 TO 6
    SWITCH nCounterModels
	  CASE 1
	    nTyp = nMODEL1
	  CASE 2
	    nTyp = nMODEL2
	  CASE 3
	    nTyp = nMODEL3
	  CASE 4
	    nTyp = nMODEL4
	  CASE 5
	    nTyp = nMODEL5
     CASE 6
	    nTyp = nMODEL6
	 ENDSWITCH
    ; Modellkontrolle def. im Makro 57
    IF (nTyp <= 0) OR (nTyp == 10) OR (nTyp == 20) OR ((nTyp >= 30) AND (nTyp <= 39)) OR (nTyp > 42) THEN
       ;
    ELSE
      BA_PRC_ModOn[nTyp] = TRUE
    ENDIF
   ENDFOR
END
;
  ;ENDFOLD (Model-Init)
;
  ;FOLD Frame-Init
;
DEF PRC_FrameInit(nMINMAX:IN,nTRANSROT:IN,rXLIMIT:IN,rYLIMIT:IN,rZLIMIT:IN,nRESERVE:IN) ; VF Limits (Mehrfach Aufruf erlaubt)
INT nMINMAX ;    Grenze    0=Minimalgrenze / 1=Maximalgrenze
INT nTRANSROT ;  Trans/Rot 0=Translation   / 1=Rotation
REAL rXLIMIT ;   X-Limit/A-Limit
REAL rYLIMIT ;   Y-Limit/B-Limit
REAL rZLIMIT ;   Z-Limit/C-Limit
INT nRESERVE ;   Frei
  SWITCH nMINMAX
    CASE 0 ; Minimalgrenze
	  SWITCH nTRANSROT
        CASE 0 ; Translation
	      VF_PRC_Min.X = rXLIMIT / 10
		   VF_PRC_Min.Y = rYLIMIT / 10
		   VF_PRC_Min.Z = rZLIMIT / 10
	    CASE 1 ; Rotation
	      VF_PRC_Min.A = rZLIMIT / 10
		   VF_PRC_Min.B = rYLIMIT / 10
		   VF_PRC_Min.C = rXLIMIT / 10
	    DEFAULT ; ncht definiert
	      B_PRC_MsgKri = TRUE
		   N_PRC_Ret1 = PRC_MsgErr(#NotifyMsg,1215,nTRANSROT)
      ENDSWITCH ; nTRANSROT
	CASE 1 ; Maximalgrenze
	  SWITCH nTRANSROT
        CASE 0 ; Translation
	      VF_PRC_Max.X = rXLIMIT / 10
		   VF_PRC_Max.Y = rYLIMIT / 10
		   VF_PRC_Max.Z = rZLIMIT / 10
	    CASE 1 ; Rotation
	      VF_PRC_Max.A = rZLIMIT / 10
		   VF_PRC_Max.B = rYLIMIT / 10
		   VF_PRC_Max.C = rXLIMIT / 10
	    DEFAULT ; ncht definiert
	      B_PRC_MsgKri = TRUE
		   N_PRC_Ret1 = PRC_MsgErr(#NotifyMsg,1216,nTRANSROT)
      ENDSWITCH ; nTRANSROT
	DEFAULT ; ncht definiert
	  B_PRC_MsgKri = TRUE
	  N_PRC_Ret1 = PRC_MsgErr(#NotifyMsg,1217,nMINMAX)
  ENDSWITCH ; nMINMAX
END
;
  ;ENDFOLD (Frame-Init)
;
  ;FOLD Default-Init
;
DEF PRC_DefaultInit() ; Setzt default Werte
INT nCounterFlags
  ; Toolkalibrier-Modus = ToolFinder
  N_PRC_SubSystem = 0
  ; Nicht Conveyor-Tech
  B_PRC_CoTech = FALSE
  ; Alive-Bit
  B_PRC_UseFct = FALSE
  ; Korr-Base 31
  N_PRC_KorBas = 31
  ; VFNr fuer Robotertausch
  N_PRC_VFNr = 1
  ; Timeout am Messpunkt [ms]
  N_PRC_TmMP = 5000
  ; Timeout bei Kommunikation [ms]
  N_PRC_TmCom = 5000
  ;Interrupt fuer RobMove
  N_PRC_Int1 = 20
  ;Interrupt fuer RobNoMove
  N_PRC_Int2 = 21
  ; Frame Max/Min
  VF_PRC_Max = {X 10.0,Y 10.0,Z 10.0,A 1.0,B 1.0,C 1.0}
  VF_PRC_Min = {X -10.0,Y -10.0,Z -10.0,A -1.0,B -1.0,C -1.0}
  ; Modellkontrolle def. im Makro 57
  ; Modellflags Aus
  FOR nCounterFlags = 1 TO 29
    IF (nCounterFlags <> 10) AND (nCounterFlags <> 20) THEN
      BA_PRC_ModOn[nCounterFlags] = FALSE
    ENDIF
    BA_PRC_ModOn[40] = FALSE
    BA_PRC_ModOn[41] = FALSE
    BA_PRC_ModOn[42] = FALSE
  ENDFOR ; nCounterFlags
  ; Fehlerflags Aus
  FOR nCounterFlags = N_PRC_FiErr TO (N_PRC_FiErr + N_PRC_LgErr - 1)
    $FLAG[nCounterFlags] = FALSE
  ENDFOR ; nCounterFlags
END
;
  ;ENDFOLD (Default-Init)
;
  ;FOLD Kommunikations Routinen
;
DEF PRC_SendeKanalOeffnen()
INT nComTimerStart
  nComTimerStart = $Rob_Timer
  WAIT FOR (NOT(I_PRC_DaSend) OR (($Rob_Timer - nComTimerStart) > N_PRC_TmCom))
  IF (($Rob_Timer - nComTimerStart) > N_PRC_TmCom) THEN
    B_PRC_MsgFlg = TRUE
    N_PRC_Err1   = N_PRC_MsgOff + 1   ; Timeout beim PRC_SendeKanalOeffnen
  ELSE
    N_PRC_Err1   = N_PRC_MsgOff
    O_PRC_DaSend = TRUE
    B_PRC_MsgFlg = FALSE
  ENDIF
END
;
DEFFCT BOOL PRC_DatenSenden()
INT nComTimerStart
  N_PRC_Err1  = N_PRC_MsgOff
  O_PRC_DaNew = TRUE
  nComTimerStart = $Rob_Timer
  WAIT FOR (I_PRC_DaAck OR (($Rob_Timer - nComTimerStart) > N_PRC_TmCom))
  IF (($Rob_Timer - nComTimerStart) > N_PRC_TmCom) THEN
    N_PRC_Err1   = N_PRC_MsgOff + 17   ; timeout beim PRC_DatenSenden
    GOTO FctErr
  ENDIF
  IF NOT((I_PRC_Data1==O_PRC_Data1) OR (I_PRC_Data2==O_PRC_Data2) OR (I_PRC_Data3==O_PRC_Data3) OR (I_PRC_Data4==O_PRC_Data4) OR (I_PRC_Data5==O_PRC_Data5) OR (I_PRC_Data6==O_PRC_Data6)) THEN
    N_PRC_Err1 = N_PRC_MsgOff + 18   ; Daten und gespiegelte daten nicht gleich beim PRC_DatenSenden
    GOTO FctErr
  ENDIF
  O_PRC_DaNew = FALSE
  nComTimerStart = $Rob_Timer
  WAIT FOR (NOT(I_PRC_DaAck) OR (($Rob_Timer - nComTimerStart) > N_PRC_TmCom))
  O_PRC_Data1 = 0
  O_PRC_Data2 = 0
  O_PRC_Data3 = 0
  O_PRC_Data4 = 0
  O_PRC_Data5 = 0
  O_PRC_Data6 = 0
  IF (($Rob_Timer - nComTimerStart) > N_PRC_TmCom) THEN
    N_PRC_Err1 = N_PRC_MsgOff + 17   ; timeout beim PRC_DatenSenden
    GOTO FctErr
  ENDIF
  RETURN(TRUE)
FctErr:
  O_PRC_DaNew  = FALSE
  O_PRC_DaSend = FALSE
  B_PRC_MsgFlg = TRUE
  RETURN(FALSE)
ENDFCT
;
DEF PRC_SendeKanalSchliessen()
INT nComTimerStart
  O_PRC_DaComp   = TRUE
  nComTimerStart = $Rob_Timer
  WAIT FOR (I_PRC_DaComp OR (($Rob_Timer - nComTimerStart) > N_PRC_TmCom))
  O_PRC_DaComp = FALSE
  O_PRC_DaSend = FALSE
  IF (($Rob_Timer - nComTimerStart) > N_PRC_TmCom) THEN
    N_PRC_Err1   = N_PRC_MsgOff + 2   ; Timeout beim warten auf I_PRC_DaComp
    B_PRC_MsgFlg = TRUE
  ELSE
    nComTimerStart = $Rob_Timer
    WAIT FOR (NOT(I_PRC_DaComp) OR (($Rob_Timer - nComTimerStart) > N_PRC_TmCom))
    IF (($Rob_Timer - nComTimerStart) > N_PRC_TmCom) THEN
      N_PRC_Err1   = N_PRC_MsgOff + 3   ; Timeout beim warten auf nicht I_PRC_DaComp
      B_PRC_MsgFlg = TRUE
    ENDIF
  ENDIF
END
;
DEFFCT BOOL PRC_EmpfangsKanalOeffnen()
INT nComTimerStart
  O_PRC_DaSend   = FALSE
  nComTimerStart = $Rob_Timer
  WAIT FOR (I_PRC_DaSend OR (($Rob_Timer - nComTimerStart) > N_PRC_TmCom))
  IF (($Rob_Timer - nComTimerStart) > N_PRC_TmCom) THEN
    N_PRC_Err1 = N_PRC_MsgOff + 26    ; Timeout beim warten auf I_PRC_DaSend
    RETURN(FALSE)
  ENDIF
  RETURN(TRUE)
ENDFCT
;
DEFFCT BOOL PRC_DatenEmpfangen ()
INT DATEN_NR
INT nComTimerStart
  DATEN_NR = 0
  REPEAT
    nComTimerStart = $Rob_Timer
    WAIT FOR (I_PRC_DaNew OR I_PRC_DaComp OR (($Rob_Timer - nComTimerStart) > N_PRC_TmCom))
    IF (($Rob_Timer - nComTimerStart) > N_PRC_TmCom) THEN
      N_PRC_Err1   = N_PRC_MsgOff + 27  ; Timeout beim warten auf I_PRC_DaNew
      B_PRC_MsgFlg = TRUE
      RETURN(FALSE)
    ENDIF
    IF I_PRC_DaNew THEN
      DATEN_NR = DATEN_NR + 1
      PRC_EmpfangsKanalLesen(DATEN_NR)
      O_PRC_DaAck    = TRUE
      nComTimerStart = $Rob_Timer
      WAIT FOR (NOT(I_PRC_DaNew) OR (($Rob_Timer - nComTimerStart) > N_PRC_TmCom))
      O_PRC_DaAck = FALSE
      IF (($Rob_Timer - nComTimerStart) > N_PRC_TmCom) THEN
        N_PRC_Err1   = N_PRC_MsgOff + 28  ; Timeout beim warten auf nicht I_PRC_DaNew
        B_PRC_MsgFlg = TRUE
        RETURN(FALSE)
      ENDIF
    ENDIF
  UNTIL I_PRC_DaComp
  RETURN(TRUE)
ENDFCT
;
DEF PRC_EmpfangsKanalLesen(DATEN_NR:IN)
INT DATEN_NR
  NA_PRC_Data[DATEN_NR,1] = I_PRC_Data1  ; Byte1
  NA_PRC_Data[DATEN_NR,2] = I_PRC_Data2  ; Byte2
  NA_PRC_Data[DATEN_NR,3] = I_PRC_Data3  ; Byte3
  NA_PRC_Data[DATEN_NR,4] = I_PRC_Data4  ; Byte4
  NA_PRC_Data[DATEN_NR,5] = I_PRC_Data5  ; Byte5
  NA_PRC_Data[DATEN_NR,6] = I_PRC_Data6  ; Byte6
  O_PRC_Data1 = NA_PRC_Data[DATEN_NR,1]  ; spiegeln Byte1
  O_PRC_Data2 = NA_PRC_Data[DATEN_NR,2]  ; spiegeln Byte2
  O_PRC_Data3 = NA_PRC_Data[DATEN_NR,3]  ; spiegeln Byte3
  O_PRC_Data4 = NA_PRC_Data[DATEN_NR,4]  ; spiegeln Byte4
  O_PRC_Data5 = NA_PRC_Data[DATEN_NR,5]  ; spiegeln Byte5
  O_PRC_Data6 = NA_PRC_Data[DATEN_NR,6]  ; spiegeln Byte6
END
;
DEF PRC_EmpfKanalSchliessen()
INT nComTimerStart
  O_PRC_Data1    = 0
  O_PRC_Data2    = 0
  O_PRC_Data3    = 0
  O_PRC_Data4    = 0
  O_PRC_Data5    = 0
  O_PRC_Data6    = 0
  O_PRC_DaComp   = TRUE
  nComTimerStart = $Rob_Timer
  WAIT FOR (NOT(I_PRC_DaComp) OR (($Rob_Timer - nComTimerStart) > N_PRC_TmCom))
  O_PRC_DaComp = FALSE
  IF (($Rob_Timer - nComTimerStart) > N_PRC_TmCom) THEN
    ; hier keine Fehlermeldung!!
  ENDIF
END
;
DEF PRC_EmpfDatenAuswerten()
  N_PRC_KennAck = NA_PRC_Data[1,2]
  N_PRC_IDAck   = NA_PRC_Data[1,1]
  N_PRC_P1Ack   = NA_PRC_Data[1,4] * 255 + NA_PRC_Data[1,3]
  N_PRC_P2Ack   = NA_PRC_Data[1,6] * 255 + NA_PRC_Data[1,5]
  PRC_ConvBytes2Real(NA_PRC_Data[2,1],NA_PRC_Data[2,2],NA_PRC_Data[2,3],NA_PRC_Data[2,4],VF_PRC_Sen.X)
  PRC_ConvBytes2Real(NA_PRC_Data[2,5],NA_PRC_Data[2,6],NA_PRC_Data[3,1],NA_PRC_Data[3,2],VF_PRC_Sen.Y)
  PRC_ConvBytes2Real(NA_PRC_Data[3,3],NA_PRC_Data[3,4],NA_PRC_Data[3,5],NA_PRC_Data[3,6],VF_PRC_Sen.Z)
  PRC_ConvBytes2Real(NA_PRC_Data[4,1],NA_PRC_Data[4,2],NA_PRC_Data[4,3],NA_PRC_Data[4,4],VF_PRC_Sen.A)
  PRC_ConvBytes2Real(NA_PRC_Data[4,5],NA_PRC_Data[4,6],NA_PRC_Data[5,1],NA_PRC_Data[5,2],VF_PRC_Sen.B)
  PRC_ConvBytes2Real(NA_PRC_Data[5,3],NA_PRC_Data[5,4],NA_PRC_Data[5,5],NA_PRC_Data[5,6],VF_PRC_Sen.C)
END
;
DEF  PRC_ConvBytes2Real (nVal4 :IN,nVal3 :IN,nVal2 :IN,nVal1 :IN,rVal :OUT )
REAL rVal
INT  nVal1
INT  nVal2
INT  nVal3
INT  nVal4
BOOL NEG
  NEG = FALSE
  IF nVal1 > 127 THEN
    nVal1 = 255 - nVal1
    nVal2 = 255 - nVal2
    nVal3 = 255 - nVal3
    nVal4 = 255 - nVal4
    NEG = TRUE
  ENDIF
  rVal = nVal1
  rVal = rVal * 256 + nVal2
  rVal = rVal * 256 + nVal3
  rVal = rVal * 256 + nVal4
  IF NEG THEN
    rVal =-(rVal + 1)
  ENDIF
  rVal = rVal / 100000
END
;
DEF PRC_ConvWort2Byte(NWORD:IN,nByte1:OUT,nByte2:OUT)
INT NWORD
INT nByte1
INT nByte2
  nByte1 = (NWORD B_AND 65280) / 256
  nByte2 =  NWORD B_AND 255
END
;
DEF  PRC_ConvReal2Bytes (rVal :IN,nVal1 :OUT,nVal2 :OUT,nVal3 :OUT,nVal4 :OUT )
REAL rVal
INT  nVal1
INT  nVal2
INT  nVal3
INT  nVal4
INT  nDWort
  nDWort = rVal * 100000
  IF rVal < 0 THEN
   if nDWort < 0 then
     nDWort = (-1* nDWort) -1
   else
     nDWort = nDWort - 1
   endif
;alt2    nDWort = sqrt(nDWort*nDWort) -1
;   nDWort = ABS(nDWort) - 1
  ENDIF
  nVal4  = nDWort B_AND 255
  nDWort = nDWort / 256
  nVal3  = nDWort B_AND 255
  nDWort = nDWort / 256
  nVal2  = nDWort B_AND 255
  nDWort = nDWort / 256
  nVal1  = nDWort B_AND 255
  nDWort = nDWort / 256
  IF nDWort >= 1 THEN
    ;Wert zu gross
  ENDIF
  IF rVal < 0 THEN
    nVal1 = 255 - nVal1
    nVal2 = 255 - nVal2
    nVal3 = 255 - nVal3
    nVal4 = 255 - nVal4
  ENDIF
END
;
DEF  PRC_Send3Real (rVal01 :IN,rVal02 :IN,rVal03 :IN )
REAL rVal01
REAL rVal02
REAL rVal03
INT  nByte01
INT  nByte02
INT  nByte03
INT  nByte04
INT  nByte05
INT  nByte06
INT  nByte07
INT  nByte08
INT  nByte09
INT  nByte10
INT  nByte11
INT  nByte12
  PRC_ConvReal2Bytes(rVal01,nByte01,nByte02,nByte03,nByte04 )
  PRC_ConvReal2Bytes(rVal02,nByte05,nByte06,nByte07,nByte08 )
  PRC_ConvReal2Bytes(rVal03,nByte09,nByte10,nByte11,nByte12 )
  PRC_Send6Byte(nByte01,nByte02,nByte03,nByte04,nByte05,nByte06 )
  PRC_Send6Byte(nByte07,nByte08,nByte09,nByte10,nByte11,nByte12 )
END
;
DEF  PRC_Send6Byte (nVal01 :IN,nVal02 :IN,nVal03 :IN,nVal04 :IN,nVal05 :IN,nVal06 :IN )
INT nVal01
INT nVal02
INT nVal03
INT nVal04
INT nVal05
INT nVal06
INT nComTimerStart
  O_PRC_Data1 = nVal02
  O_PRC_Data2 = nVal01
  O_PRC_Data3 = nVal04
  O_PRC_Data4 = nVal03
  O_PRC_Data5 = nVal06
  O_PRC_Data6 = nVal05
; DEFFCT BOOL PRC_DatenSenden()
  N_PRC_Err1  = N_PRC_MsgOff
  O_PRC_DaNew = TRUE
  nComTimerStart = $Rob_Timer
  WAIT FOR (I_PRC_DaAck OR (($Rob_Timer - nComTimerStart) > N_PRC_TmCom))
  IF (($Rob_Timer - nComTimerStart) > N_PRC_TmCom) THEN
    N_PRC_Err1   = N_PRC_MsgOff + 17   ; timeout beim PRC_DatenSenden
    GOTO DataSendErr
  ENDIF
  IF NOT((I_PRC_Data1==O_PRC_Data1) OR (I_PRC_Data2==O_PRC_Data2) OR (I_PRC_Data3==O_PRC_Data3) OR (I_PRC_Data4==O_PRC_Data4) OR (I_PRC_Data5==O_PRC_Data5) OR (I_PRC_Data6==O_PRC_Data6)) THEN
    N_PRC_Err1 = N_PRC_MsgOff + 18   ; Daten und gespiegelte daten nicht gleich beim PRC_DatenSenden
    GOTO DataSendErr
  ENDIF
  O_PRC_DaNew = FALSE
  nComTimerStart = $Rob_Timer
  WAIT FOR (NOT(I_PRC_DaAck) OR (($Rob_Timer - nComTimerStart) > N_PRC_TmCom))
  O_PRC_Data1 = 0
  O_PRC_Data2 = 0
  O_PRC_Data3 = 0
  O_PRC_Data4 = 0
  O_PRC_Data5 = 0
  O_PRC_Data6 = 0
  IF (($Rob_Timer - nComTimerStart) > N_PRC_TmCom) THEN
    N_PRC_Err1 = N_PRC_MsgOff + 17   ; timeout beim PRC_DatenSenden
    GOTO DataSendErr
  ENDIF
  RETURN
DataSendErr:
  O_PRC_DaNew  = FALSE
  O_PRC_DaSend = FALSE
  B_PRC_MsgFlg = TRUE
  RETURN
END
;
DEF PRC_SendInfo (nID:IN,nPar1:IN,nPar2:IN,nPar3:IN,nPar4:IN)
INT  nID
INT  nPar1
INT  nPar2
INT  nPar3
INT  nPar4
INT  nByte1
INT  nByte2
INT  nByte01
INT  nByte02
INT  nByte03
INT  nByte04
INT  nByte05
INT  nByte06
INT  nByte07
INT  nByte08
INT  nByte09
INT  nByte10
INT  nByte11
INT  nByte12
   PRC_SendeKanalOeffnen()
   IF N_PRC_Err1 == N_PRC_MsgOff THEN
      IF varState("nPar3") <> #INITIALIZED THEN ; Sende Poseinfo (3)
  	      O_PRC_Data2 = N_PRC_Specf
         O_PRC_Data1 = nID
         PRC_ConvWort2Byte(nPar1,nByte1,nByte2)   ; Modell HL Byte gedreht!!!
         O_PRC_Data3 = nByte2
         O_PRC_Data4 = nByte1
         PRC_ConvWort2Byte(nPar2,nByte1,nByte2)   ; Sequenz HL Byte gedreht!!!
         O_PRC_Data5 = nByte2
         O_PRC_Data6 = nByte1
	   ELSE ; Sende Pose ID (13)
	      O_PRC_Data2 = N_PRC_Specf
         O_PRC_Data1 = nID
	      PRC_ConvWort2Byte(nPar1,nByte1,nByte2)   ; Modell HL Byte gedreht!!!
         O_PRC_Data3 = nByte2
         O_PRC_Data4 = nByte1
         PRC_ConvWort2Byte(nPar2,nByte1,nByte2)   ; Sequenz HL Byte gedreht!!!
         O_PRC_Data5 = nByte2
         O_PRC_Data6 = nByte1
	      IF NOT PRC_DatenSenden() THEN
            RETURN
         ENDIF
	      O_PRC_Data2 = N_PRC_Specf
         O_PRC_Data1 = nID
	      PRC_ConvWort2Byte(nPar3,nByte1,nByte2)   ; Frame-ID HL Byte gedreht!!!
         O_PRC_Data3 = nByte2
         O_PRC_Data4 = nByte1
         PRC_ConvWort2Byte(nPar4,nByte1,nByte2)   ; Tool-ID HL Byte gedreht!!!
         O_PRC_Data5 = nByte2
         O_PRC_Data6 = nByte1
      ENDIF
	   IF NOT PRC_DatenSenden() THEN
         RETURN
      ENDIF
      ;PRC_Send3Real($POS_ACT.X,$POS_ACT.Y,$POS_ACT.Z )
      PRC_ConvReal2Bytes($POS_ACT.X,nByte01,nByte02,nByte03,nByte04 )
      PRC_ConvReal2Bytes($POS_ACT.Y,nByte05,nByte06,nByte07,nByte08 )
      PRC_ConvReal2Bytes($POS_ACT.Z,nByte09,nByte10,nByte11,nByte12 )
      PRC_Send6Byte(nByte01,nByte02,nByte03,nByte04,nByte05,nByte06 )
      PRC_Send6Byte(nByte07,nByte08,nByte09,nByte10,nByte11,nByte12 )
      ;PRC_Send3Real($POS_ACT.A,$POS_ACT.B,$POS_ACT.C )
      PRC_ConvReal2Bytes($POS_ACT.A,nByte01,nByte02,nByte03,nByte04 )
      PRC_ConvReal2Bytes($POS_ACT.B,nByte05,nByte06,nByte07,nByte08 )
      PRC_ConvReal2Bytes($POS_ACT.C,nByte09,nByte10,nByte11,nByte12 )
      PRC_Send6Byte(nByte01,nByte02,nByte03,nByte04,nByte05,nByte06 )
      PRC_Send6Byte(nByte07,nByte08,nByte09,nByte10,nByte11,nByte12 )
      ;PRC_Send3Real($AXIS_ACT.A1,$AXIS_ACT.A2,$AXIS_ACT.A3 )
      PRC_ConvReal2Bytes($AXIS_ACT.A1,nByte01,nByte02,nByte03,nByte04 )
      PRC_ConvReal2Bytes($AXIS_ACT.A2,nByte05,nByte06,nByte07,nByte08 )
      PRC_ConvReal2Bytes($AXIS_ACT.A3,nByte09,nByte10,nByte11,nByte12 )
      PRC_Send6Byte(nByte01,nByte02,nByte03,nByte04,nByte05,nByte06 )
      PRC_Send6Byte(nByte07,nByte08,nByte09,nByte10,nByte11,nByte12 )
      ;PRC_Send3Real($AXIS_ACT.A4,$AXIS_ACT.A5,$AXIS_ACT.A6 )
      PRC_ConvReal2Bytes($AXIS_ACT.A4,nByte01,nByte02,nByte03,nByte04 )
      PRC_ConvReal2Bytes($AXIS_ACT.A5,nByte05,nByte06,nByte07,nByte08 )
      PRC_ConvReal2Bytes($AXIS_ACT.A6,nByte09,nByte10,nByte11,nByte12 )
      PRC_Send6Byte(nByte01,nByte02,nByte03,nByte04,nByte05,nByte06 )
      PRC_Send6Byte(nByte07,nByte08,nByte09,nByte10,nByte11,nByte12 )
      IF ($ACT_BASE == 11) AND(B_PRC_CoTech == TRUE) THEN ; Base lesen waehrend Conveyorfahrt
         VF_PRC_ConTmp   = $NULLFRAME
         VF_PRC_SenPrea  = $NULLFRAME
         VF_PRC_ConTmp.x = $SEN_PREA_C[1]
         VF_PRC_SenPrea=BASE_DATA[11]:VF_PRC_ConTmp
         ;PRC_Send3Real(VF_PRC_SenPrea.X,VF_PRC_SenPrea.Y,VF_PRC_SenPrea.Z )
         PRC_ConvReal2Bytes(VF_PRC_SenPrea.X,nByte01,nByte02,nByte03,nByte04 )
         PRC_ConvReal2Bytes(VF_PRC_SenPrea.Y,nByte05,nByte06,nByte07,nByte08 )
         PRC_ConvReal2Bytes(VF_PRC_SenPrea.Z,nByte09,nByte10,nByte11,nByte12 )
         PRC_Send6Byte(nByte01,nByte02,nByte03,nByte04,nByte05,nByte06 )
         PRC_Send6Byte(nByte07,nByte08,nByte09,nByte10,nByte11,nByte12 )
         ;PRC_Send3Real(VF_PRC_SenPrea.A,VF_PRC_SenPrea.B,VF_PRC_SenPrea.C )
         PRC_ConvReal2Bytes(VF_PRC_SenPrea.A,nByte01,nByte02,nByte03,nByte04 )
         PRC_ConvReal2Bytes(VF_PRC_SenPrea.B,nByte05,nByte06,nByte07,nByte08 )
         PRC_ConvReal2Bytes(VF_PRC_SenPrea.C,nByte09,nByte10,nByte11,nByte12 )
         PRC_Send6Byte(nByte01,nByte02,nByte03,nByte04,nByte05,nByte06 )
         PRC_Send6Byte(nByte07,nByte08,nByte09,nByte10,nByte11,nByte12 )
         ;PRC_Send3Real($TOOL.X,$TOOL.Y,$TOOL.Z )
         PRC_ConvReal2Bytes($TOOL.X,nByte01,nByte02,nByte03,nByte04 )
         PRC_ConvReal2Bytes($TOOL.Y,nByte05,nByte06,nByte07,nByte08 )
         PRC_ConvReal2Bytes($TOOL.Z,nByte09,nByte10,nByte11,nByte12 )
         PRC_Send6Byte(nByte01,nByte02,nByte03,nByte04,nByte05,nByte06 )
         PRC_Send6Byte(nByte07,nByte08,nByte09,nByte10,nByte11,nByte12 )
         ;PRC_Send3Real($TOOL.A,$TOOL.B,$TOOL.C )
         PRC_ConvReal2Bytes($TOOL.A,nByte01,nByte02,nByte03,nByte04 )
         PRC_ConvReal2Bytes($TOOL.B,nByte05,nByte06,nByte07,nByte08 )
         PRC_ConvReal2Bytes($TOOL.C,nByte09,nByte10,nByte11,nByte12 )
         PRC_Send6Byte(nByte01,nByte02,nByte03,nByte04,nByte05,nByte06 )
         PRC_Send6Byte(nByte07,nByte08,nByte09,nByte10,nByte11,nByte12 )
      ELSE
         ;PRC_Send3Real($BASE.X,$BASE.Y,$BASE.Z )
         PRC_ConvReal2Bytes($BASE.X,nByte01,nByte02,nByte03,nByte04 )
         PRC_ConvReal2Bytes($BASE.Y,nByte05,nByte06,nByte07,nByte08 )
         PRC_ConvReal2Bytes($BASE.Z,nByte09,nByte10,nByte11,nByte12 )
         PRC_Send6Byte(nByte01,nByte02,nByte03,nByte04,nByte05,nByte06 )
         PRC_Send6Byte(nByte07,nByte08,nByte09,nByte10,nByte11,nByte12 )
         ;PRC_Send3Real($BASE.A,$BASE.B,$BASE.C )
         PRC_ConvReal2Bytes($BASE.A,nByte01,nByte02,nByte03,nByte04 )
         PRC_ConvReal2Bytes($BASE.B,nByte05,nByte06,nByte07,nByte08 )
         PRC_ConvReal2Bytes($BASE.C,nByte09,nByte10,nByte11,nByte12 )
         PRC_Send6Byte(nByte01,nByte02,nByte03,nByte04,nByte05,nByte06 )
         PRC_Send6Byte(nByte07,nByte08,nByte09,nByte10,nByte11,nByte12 )
         ;PRC_Send3Real($TOOL.X,$TOOL.Y,$TOOL.Z )
         PRC_ConvReal2Bytes($TOOL.X,nByte01,nByte02,nByte03,nByte04 )
         PRC_ConvReal2Bytes($TOOL.Y,nByte05,nByte06,nByte07,nByte08 )
         PRC_ConvReal2Bytes($TOOL.Z,nByte09,nByte10,nByte11,nByte12 )
         PRC_Send6Byte(nByte01,nByte02,nByte03,nByte04,nByte05,nByte06 )
         PRC_Send6Byte(nByte07,nByte08,nByte09,nByte10,nByte11,nByte12 )
         ;PRC_Send3Real($TOOL.A,$TOOL.B,$TOOL.C )
         PRC_ConvReal2Bytes($TOOL.A,nByte01,nByte02,nByte03,nByte04 )
         PRC_ConvReal2Bytes($TOOL.B,nByte05,nByte06,nByte07,nByte08 )
         PRC_ConvReal2Bytes($TOOL.C,nByte09,nByte10,nByte11,nByte12 )
         PRC_Send6Byte(nByte01,nByte02,nByte03,nByte04,nByte05,nByte06 )
         PRC_Send6Byte(nByte07,nByte08,nByte09,nByte10,nByte11,nByte12 )
      ENDIF
      PRC_SendeKanalSchliessen()
   ENDIF
END
;
  ;ENDFOLD (Kommunikations Routinen)
;
  ;FOLD CheckMaxVF
;
DEFFCT  BOOL PRC_CheckMaxVF(BP :IN)
FRAME BP
  IF ((BP.X<=VF_PRC_Max.X) AND (BP.Y<=VF_PRC_Max.Y) AND (BP.Z<=VF_PRC_Max.Z) AND (BP.A<=VF_PRC_Max.A) AND (BP.B<=VF_PRC_Max.B) AND (BP.C<=VF_PRC_Max.C)) THEN
    IF ((BP.X>=VF_PRC_Min.X) AND (BP.Y>=VF_PRC_Min.Y) AND (BP.Z>=VF_PRC_Min.Z) AND (BP.A>=VF_PRC_Min.A) AND (BP.B>=VF_PRC_Min.B) AND (BP.C>=VF_PRC_Min.C)) THEN
      RETURN  (TRUE)
    ELSE
      N_PRC_Err1 = 1019
      RETURN(FALSE)
    ENDIF
  ELSE
    N_PRC_Err1 = 1020
    RETURN  (FALSE)
  ENDIF
ENDFCT
  ;ENDFOLD (CheckMaxVF)
;
  ;FOLD CheckParameter
;
DEFFCT INT PRC_CheckParams(nTYP:IN,nSUBTYP:IN,nNR:IN,nPAR1:IN,nPAR2:IN,nPAR3:IN,nPAR4:IN)
INT nTYP
INT nSUBTYP
INT nNR
INT nPAR1
INT nPAR2
INT nPAR3
INT nPAR4
  IF ((nTYP < 0) OR (nTYP > 255)) THEN
    RETURN(904)   ;USER-PAR2 ungueltig (0 - 255)      z.B. Modellnummer
  ENDIF
  IF ((nSUBTYP < 0) OR (nSUBTYP > 65535)) THEN
    RETURN(905)   ;USER-PAR3 ungueltig (0 - 65535)    Z.B. Routine
  ENDIF
  IF ((nNR < -180) OR (nNR > 65535)) THEN
    RETURN(906)   ;USER-PAR4 ungueltig (-180 - 65535)    z.B. Punkt Nr./X-Limit
  ENDIF
  IF (nPAR1 < -180) OR (nPAR1 >255) THEN
    RETURN(907)   ;USER-PAR5 ungueltig (-180 - 255)   z.B. Y-Limit
  ENDIF
  IF (nPAR2 < -180) OR (nPAR2 >255) THEN
    RETURN(907)   ;USER-PAR6 ungueltig (-180 - 255)   z.B. Z-Limit
  ENDIF
  RETURN(0)
ENDFCT
;
  ;ENDFOLD (CheckParameter)
;
  ;FOLD PRC_DebugDlg
;
DEF PRC_DebugDlg(nNr:IN,rPar1:IN,rPar2:IN)
INT  nNr
INT  nPar1
INT  nPar2
REAL rPar1
REAL rPar2
  IF varState("rPar1") <> #Initialized THEN
    rPar1 = 0
  ENDIF
  IF varState("rPar2") <> #Initialized THEN
    rPar2 = 0
  ENDIF
  nPar1 = rPar1
  nPar2 = rPar2
  IF (B_PRC_Debug == TRUE) AND (($mode_op == #T1) OR ($mode_op == #T2)) THEN
    B_PRC_MsgKri = TRUE
    IF B_PRC_DebugH THEN
      N_PRC_Ret1 = PRC_MsgErr(#DlgMsg,nNr,nPar1,nPar2)
    ELSE
      N_PRC_Ret1 = PRC_MsgErr(#NotifyMsg,nNr,nPar1,nPar2)
    ENDIF
  ENDIF
  IF B_PRC_DebugH THEN
    HALT
  ENDIF
END
;
  ;ENDFOLD (PRC_DebugDlg)
;
  ;FOLD Ausgabe Roboter bewegt sich an Perceptron
;
DEF PRC_Move(PRC_Move: IN)
INT PRC_Move
  SWITCH PRC_Move
    CASE 1
      O_PRC_RobBwg = TRUE
    CASE 2
      O_PRC_RobBwg = FALSE
  ENDSWITCH
END
;
  ;ENDFOLD (Ausgabe Roboter bewegt sich an Perceptron)
;
    ;ENDFOLD (Perceptron Lokale Unterprogramme)
;
;Meldungsart:
;In Automatik duerfen nur NIO-Meldungen ausgegeben werden
;In Single-Step alle wichtigen Meldungen
;In Single-Step + Debugger-Flag alle Meldungen
;
;FOLD Perceptron Meldungen
DEFFCT INT PRC_MsgErr (MSG_TYP:IN, MSG_NR:IN, rPar :IN, nPar:IN)
DECL Real          rPar
DECL INT           MSG_NR
DECL INT           nPar
DECL INT           OFFSET
DECL PRC_MsgType   MSG_TYP
DECL STATE_T       STATE
DECL KRLMSG_T      USER_MSG
DECL KRLMSGPAR_T   PAR[3]
DECL KRLMSGOPT_T   OPT
DECL KrlMsgDlgSK_T SK[7]
DECL Char          sMeldFunction[80]
DECL INT           nTmp
DECL INT           nDlgHandle
DECL INT           nDlgAnswer
  IF ($mode_op <> #T1) AND ($mode_op <> #T2) AND (NOT B_PRC_MsgKri) THEN
    RETURN(1)
  ENDIF
  B_PRC_MsgKri = FALSE
  IF (MSG_NR == 0) OR (MSG_NR == 50) OR (MSG_NR == 100) OR (MSG_NR == 200) OR (MSG_NR == 250) OR (MSG_NR == 300) OR (MSG_NR == 400) OR (MSG_NR == 500) OR (MSG_NR == 600) OR (MSG_NR == 700) OR (MSG_NR == 800) OR (MSG_NR == 900) OR (MSG_NR == 1000) OR (MSG_NR == 1100) OR (MSG_NR == 1200) THEN
    IF B_PRC_Debug == FALSE THEN
      RETURN(1)
    ENDIF
  ENDIF
;
;FOLD Init
;
  IF varState("rPar") <> #INITIALIZED THEN
  	 rPar = -1
  ENDIF
  IF varState("nPar") <> #INITIALIZED THEN
  	 nPar = -1
  ENDIF
  USER_MSG         = { Modul[] "PRC_MsgErr", Nr 1, Msg_txt[] " "}
  Par[1]           = { Par_type #Value, Par_txt[] " " }
  Opt              = { VL_Stop TRUE, Clear_P_Reset TRUE, Log_To_DB TRUE }
  FOR nTmp = 1 TO 7
    SK[nTmp] = {Sk_Type #Empty}
  ENDFOR
;
;ENDFOLD (Init)
;
;FOLD Fehler Funktion
;
  sMeldFunction[] = "Unbekannt - "
  IF ((MSG_NR >= 1) AND (MSG_NR <= 49)) THEN
  	sMeldFunction[] = "Debug - "
  ENDIF
  IF ((MSG_NR >= 50) AND (MSG_NR <= 99)) THEN
  	sMeldFunction[] = "Sync - "
  ENDIF
  IF ((MSG_NR >= 100) AND (MSG_NR <= 199)) THEN
  	sMeldFunction[] = "Messstart - "
  ENDIF
  IF ((MSG_NR >= 200) AND (MSG_NR <= 249)) THEN
  	sMeldFunction[] = "Punktmessung - "
  ENDIF
  IF ((MSG_NR >= 250) AND (MSG_NR <= 299)) THEN
  	sMeldFunction[] = "Scanning - "
  ENDIF
  IF ((MSG_NR >= 300) AND (MSG_NR <= 399)) THEN
  	sMeldFunction[] = "Statusanforderung - "
  ENDIF
  IF ((MSG_NR >= 400) AND (MSG_NR <= 499)) THEN
  	sMeldFunction[] = "Messende - "
  ENDIF
  IF ((MSG_NR >= 500) AND (MSG_NR <= 599)) THEN
  	sMeldFunction[] = "Reset - "
  ENDIF
  IF ((MSG_NR >= 600) AND (MSG_NR <= 699)) THEN
  	sMeldFunction[] = "Sensortausch - "
  ENDIF
  IF ((MSG_NR >= 700) AND (MSG_NR <= 799)) THEN
  	sMeldFunction[] = "Robotertausch - "
  ENDIF
  IF ((MSG_NR >= 800) AND (MSG_NR <= 899)) THEN
  	sMeldFunction[] = "Hole UP-Nr - "
  ENDIF
  IF ((MSG_NR >= 900) AND (MSG_NR <= 999)) THEN
  	sMeldFunction[] = "Ungueltige Parameter - "
  ENDIF
  IF ((MSG_NR >= 1000) AND (MSG_NR <= 1099)) THEN
  	sMeldFunction[] = "Hole Korrektur - "
  ENDIF
  IF ((MSG_NR >= 1100) AND (MSG_NR <= 1199)) THEN
  	sMeldFunction[] = "Alarme - "
  ENDIF
  IF ((MSG_NR >= 1200) AND (MSG_NR <= 1299)) THEN
  	sMeldFunction[] = "Init - "
  ENDIF
  IF (MSG_NR == 9000) THEN
  	sMeldFunction[] = "Version - "
  ENDIF
;
;FOLD (Fehler Funktion)
;
;FOLD Meldungs-Nr
;
  OFFSET  = 0
  nTmp    = rPar
  SK[1]   = {Sk_Type #Value,Sk_Txt[] "Weiter"}
  SWITCH MSG_NR
;	Fehler (Debug)
    CASE 1
      swrite(USER_MSG.MSG_TXT[],STATE,OFFSET,"Status %d",nTmp)
      SK[1] = {Sk_Type #Value,Sk_Txt[] "OK"}
    CASE 2
      swrite(USER_MSG.MSG_TXT[],STATE,OFFSET,"Modell %d",nTmp)
      SK[1] = {Sk_Type #Value,Sk_Txt[] "OK"}
    CASE 3
      swrite(USER_MSG.MSG_TXT[],STATE,OFFSET,"Punkt %d",nTmp)
      SK[1] = {Sk_Type #Value,Sk_Txt[] "OK"}
    CASE 4
      USER_MSG.MSG_TXT[] = "Messende"
      SK[1] = {Sk_Type #Value,Sk_Txt[] "OK"}
    CASE 5
      USER_MSG.MSG_TXT[] = "Sensortausch"
      SK[1] = {Sk_Type #Value,Sk_Txt[] "OK"}
    CASE 6
      USER_MSG.MSG_TXT[] = "StartMessung"
      SK[1] = {Sk_Type #Value,Sk_Txt[] "OK"}
    CASE 7
      USER_MSG.MSG_TXT[] = "Korrekturwerte holen"
      SK[1] = {Sk_Type #Value,Sk_Txt[] "OK"}
    CASE 8
      USER_MSG.MSG_TXT[] = "Korrekturwerte setzen"
      SK[1] = {Sk_Type #Value,Sk_Txt[] "OK"}
    CASE 9
      USER_MSG.MSG_TXT[] = "System Reset"
      SK[1] = {Sk_Type #Value,Sk_Txt[] "OK"}
    CASE 10
      USER_MSG.MSG_TXT[] = "Robotertausch"
      SK[1] = {Sk_Type #Value,Sk_Txt[] "OK"}
    CASE 11
      USER_MSG.MSG_TXT[] = "Messstart von SPS"
      SK[1] = {Sk_Type #Value,Sk_Txt[] "OK"}
    CASE 16
      USER_MSG.MSG_TXT[] = "Senspruef: StartMessung"
      SK[1] = {Sk_Type #Value,Sk_Txt[] "OK"}
    CASE 23
      USER_MSG.MSG_TXT[] = "System im Kalibiriermodus"
      SK[1] = {Sk_Type #Value,Sk_Txt[] "OK"}
    CASE 24
      USER_MSG.MSG_TXT[] = "Hole UP Nr."
      SK[1] = {Sk_Type #Value,Sk_Txt[] "OK"}
    CASE 25
      swrite(USER_MSG.MSG_TXT[],STATE,OFFSET,"Modell %d , Routine %d",nTmp,nPar)
      SK[1] = {Sk_Type #Value,Sk_Txt[] "OK"}
    CASE 26
      USER_MSG.MSG_TXT[] = "Toolfinder: StartMessung"
      SK[1] = {Sk_Type #Value,Sk_Txt[] "OK"}
;	Fehler (Init)
    CASE 50
  		USER_MSG.MSG_TXT[] = "Erfolgreich"
    CASE 51
  		USER_MSG.MSG_TXT[] = "Timeout: Beim Sendekanal oeffnen"
      $FLAG[F_PRC_TmOut]=TRUE
    CASE 56
  		USER_MSG.MSG_TXT[] = "System im Offline/Programmier-Modus"
    CASE 57
  		USER_MSG.MSG_TXT[] = "System bereits gestartet"
    CASE 58
  		USER_MSG.MSG_TXT[] = "Fehler allgemein"
    CASE 59
  		USER_MSG.MSG_TXT[] = "Fehler nicht spezifiziert"
    CASE 67
      USER_MSG.MSG_TXT[] = "Timeout: Beim Daten Senden"
      $FLAG[F_PRC_TmOut]=TRUE
    CASE 68
      USER_MSG.MSG_TXT[] = "Daten nicht gespiegelt"
    CASE 73
      USER_MSG.MSG_TXT[] = "System im Kalibrier-Modus"
    CASE 74
      USER_MSG.MSG_TXT[] = "System im Programmier-Modus"
    CASE 77
  		USER_MSG.MSG_TXT[] = "Timeout: Beim warten auf I_PRC_DaNew"
      $FLAG[F_PRC_TmOut]=TRUE
    CASE 78
      USER_MSG.MSG_TXT[] = "Timeout: Beim warten auf nicht I_PRC_DaNew"
      $FLAG[F_PRC_TmOut]=TRUE
    CASE 79
      USER_MSG.MSG_TXT[] = "System im Basefinder-Modus"
    CASE 80
      USER_MSG.MSG_TXT[] = "System im Toolfinder-Modus"
    CASE 93
      USER_MSG.MSG_TXT[] = "Falsche Return ID"
    CASE 94
      USER_MSG.MSG_TXT[] = "Abbruch durch User"
      SK[1] = {Sk_Type #Value,Sk_Txt[] "OK"}
    CASE 95
      USER_MSG.MSG_TXT[] = "Reset durchfuehren"
      SK[2] = {Sk_Type #Value,Sk_Txt[] "Reset"}
;	Fehler (Messstart)
    CASE 100
  		USER_MSG.MSG_TXT[] = "Erfolgreich"
    CASE 101
  		USER_MSG.MSG_TXT[] = "Timeout: Beim Sendekanal oeffnen"
      $FLAG[F_PRC_TmOut]=TRUE
    CASE 102
  		USER_MSG.MSG_TXT[] = "Timeout: Beim warten auf I_PRC_DaComp"
      $FLAG[F_PRC_TmOut]=TRUE
    CASE 103
  		USER_MSG.MSG_TXT[] = "Timeout: Beim warten auf nicht I_PRC_DaComp"
      $FLAG[F_PRC_TmOut]=TRUE
    CASE 104
  		USER_MSG.MSG_TXT[] = "Timeout: Beim warten auf I_PRC_MEACK"
      $FLAG[F_PRC_TmOut]=TRUE
    CASE 105
  		USER_MSG.MSG_TXT[] = "Modell oder Routine nicht definiert"
      SK[2] = {Sk_Type #Value,Sk_Txt[] "Reset"}
    CASE 106
  		USER_MSG.MSG_TXT[] = "System im Offline/Programmier-Modus"
      SK[3] = {Sk_Type #Value,Sk_Txt[] "Wdh."}
    CASE 107
  		USER_MSG.MSG_TXT[] = "System bereits gestartet"
      SK[2] = {Sk_Type #Value,Sk_Txt[] "Reset"}
    CASE 108
  		USER_MSG.MSG_TXT[] = "Fehler allgemein"
      SK[2] = {Sk_Type #Value,Sk_Txt[] "Reset"}
    CASE 109
  		USER_MSG.MSG_TXT[] = "Fehler nicht spezifiziert"
      SK[2] = {Sk_Type #Value,Sk_Txt[] "Reset"}
    CASE 111
  		USER_MSG.MSG_TXT[] = "System mit anderem Modell gestartet"
      SK[2] = {Sk_Type #Value,Sk_Txt[] "Reset"}
    CASE 112
  		USER_MSG.MSG_TXT[] = "System von der SPS gestartet"
      SK[2] = {Sk_Type #Value,Sk_Txt[] "Reset"}
    CASE 117
  		USER_MSG.MSG_TXT[] = "Timeout: Beim Daten Senden"
      $FLAG[F_PRC_TmOut]=TRUE
    CASE 118
      USER_MSG.MSG_TXT[] = "Daten nicht gespiegelt"
    CASE 124
      USER_MSG.MSG_TXT[] = "System nicht gestartet"
    CASE 126
  		USER_MSG.MSG_TXT[] = "Timeout: Beim warten auf I_PRC_DaSend"
      $FLAG[F_PRC_TmOut]=TRUE
    CASE 127
  		USER_MSG.MSG_TXT[] = "Timeout: Beim warten auf I_PRC_DaNew"
    CASE 128
  		USER_MSG.MSG_TXT[] = "Timeout: Beim warten auf nicht I_PRC_DaNew"
      $FLAG[F_PRC_TmOut]=TRUE
    CASE 129
  		USER_MSG.MSG_TXT[] = "Routinennummer ist 0"
    CASE 135
  		USER_MSG.MSG_TXT[] = "Anzahl Messpunkte zu klein u. falsche PunktFolge"
    CASE 136
  		USER_MSG.MSG_TXT[] = "Ungueltiger PAR_1 bei Messende"
    CASE 137
  		USER_MSG.MSG_TXT[] = "Anzahl Messpunkte zu klein"
    CASE 140
      swrite(USER_MSG.MSG_TXT[],STATE,OFFSET,"UP Mod: %d/Rout: %d nicht definiert; DAT bearbeiten",nTmp,nPar)
    CASE 141
      swrite(USER_MSG.MSG_TXT[],STATE,OFFSET,"UP Mod: %d/Rout: %d ist 0; DAT bearbeiten",nTmp,nPar)
    CASE 143
      USER_MSG.MSG_TXT[] = "Falsche Return ID"
;	Fehler (Punktmessung)
    CASE 200
  		USER_MSG.MSG_TXT[] = "Erfolgreich"
    CASE 201
  		USER_MSG.MSG_TXT[] = "Timeout: Beim Sendekanal oeffnen"
      $FLAG[F_PRC_TmOut]=TRUE
    CASE 202
  		USER_MSG.MSG_TXT[] = "Timeout: Beim warten auf I_PRC_DaComp"
      $FLAG[F_PRC_TmOut]=TRUE
    CASE 203
      USER_MSG.MSG_TXT[] = "Timeout: Beim warten auf nicht I_PRC_DaComp"
      $FLAG[F_PRC_TmOut]=TRUE
    CASE 212
      USER_MSG.MSG_TXT[] = "Timeout: Beim warten auf I_PRC_Zyklus"
      $FLAG[F_PRC_TmOut]=TRUE
    CASE 213
  		USER_MSG.MSG_TXT[] = "Fehler allgemeine"
    CASE 217
      USER_MSG.MSG_TXT[] = "Timeout: Beim Daten Senden"
      $FLAG[F_PRC_TmOut]=TRUE
    CASE 218
      USER_MSG.MSG_TXT[] = "Daten nicht gespiegelt"
    CASE 223
  		USER_MSG.MSG_TXT[] = "Positionsnummer ungueltig"
    CASE 224
  		USER_MSG.MSG_TXT[] = "System nicht gestartet"
    CASE 225
  		USER_MSG.MSG_TXT[] = "Timeout: Beim warten auf I_PRC_MEACK"
      $FLAG[F_PRC_TmOut]=TRUE
    CASE 226
  		USER_MSG.MSG_TXT[] = "Timeout: Beim warten auf I_PRC_DaSend"
      $FLAG[F_PRC_TmOut]=TRUE
    CASE 227
  		USER_MSG.MSG_TXT[] = "Falsche Punktreihenfolge"
    CASE 228
      swrite(USER_MSG.MSG_TXT[],STATE,OFFSET,"Sensormontage pruefen im Punkt: %d",nPar)
      SK[2] = {Sk_Type #Value,Sk_Txt[] "Wdh."}
    CASE 229
      swrite(USER_MSG.MSG_TXT[],STATE,OFFSET,"Robotermontage pruefen im Punkt: %d",nPar)
      SK[2] = {Sk_Type #Value,Sk_Txt[] "Wdh."}
;	Fehler (Scanning)
    CASE 250
  		USER_MSG.MSG_TXT[] = "Erfolgreich"
    CASE 251
  		USER_MSG.MSG_TXT[] = "Timeout: Beim Sendekanal oeffnen"
      $FLAG[F_PRC_TmOut]=TRUE
    CASE 252
      USER_MSG.MSG_TXT[] = "Timeout: Beim warten auf I_PRC_DaComp"
      $FLAG[F_PRC_TmOut]=TRUE
    CASE 253
      USER_MSG.MSG_TXT[] = "Timeout: Beim warten auf nicht I_PRC_DaComp"
      $FLAG[F_PRC_TmOut]=TRUE
    CASE 267
      USER_MSG.MSG_TXT[] = "Timeout: Beim Daten Senden"
      $FLAG[F_PRC_TmOut]=TRUE
    CASE 268
      USER_MSG.MSG_TXT[] = "Daten nicht gespiegelt"
    CASE 281
  		USER_MSG.MSG_TXT[] = "Fehler: I_PRC_EScAck noch gesetzt"
    CASE 282
  		USER_MSG.MSG_TXT[] = "Timeout: Beim warten auf I_PRC_EScAck"
      $FLAG[F_PRC_TmOut]=TRUE
    CASE 283
  		USER_MSG.MSG_TXT[] = "Positionsnummer ungueltig"
    CASE 284
  		USER_MSG.MSG_TXT[] = "System nicht gestartet"
    CASE 285
  		USER_MSG.MSG_TXT[] = "Fehler allgemeine"
    CASE 286
  		USER_MSG.MSG_TXT[] = "Fehler nicht spezifiziert"
    CASE 291
  		USER_MSG.MSG_TXT[] = "Fehler: I_PRC_SScAck noch gesetzt"
    CASE 292
  		USER_MSG.MSG_TXT[] = "Timeout: Beim warten auf I_PRC_SScAck"
      $FLAG[F_PRC_TmOut]=TRUE
;	Fehler (Statusanforderung)
    CASE 300
  		USER_MSG.MSG_TXT[] = "Erfolgreich"
    CASE 301
  		USER_MSG.MSG_TXT[] = "Timeout: Beim Sendekanal oeffnen"
      $FLAG[F_PRC_TmOut]=TRUE
    CASE 306
  		USER_MSG.MSG_TXT[] = "System im Offline/Programmier-Modus"
    CASE 307
  		USER_MSG.MSG_TXT[] = "System bereits gestartet"
    CASE 308
  		USER_MSG.MSG_TXT[] = "Fehler allgemein"
    CASE 309
  		USER_MSG.MSG_TXT[] = "Fehler nicht spezifiziert"
    CASE 317
  		USER_MSG.MSG_TXT[] = "Timeout: Beim Daten Senden"
      $FLAG[F_PRC_TmOut]=TRUE
    CASE 318
      USER_MSG.MSG_TXT[] = "Daten nicht gespiegelt"
    CASE 323
      USER_MSG.MSG_TXT[] = "System im Kalibrier-Modus"
    CASE 324
      USER_MSG.MSG_TXT[] = "System im Programmier-Modus"
    CASE 327
  		USER_MSG.MSG_TXT[] = "Timeout: Beim warten auf I_PRC_DaNew"
      $FLAG[F_PRC_TmOut]=TRUE
    CASE 328
  		USER_MSG.MSG_TXT[] = "Timeout: Beim warten auf nicht I_PRC_DaNew"
      $FLAG[F_PRC_TmOut]=TRUE
    CASE 329
      USER_MSG.MSG_TXT[] = "System im Basefinder-Modus"
    CASE 330
      USER_MSG.MSG_TXT[] = "System im Toolfinder-Modus"
    CASE 343
      USER_MSG.MSG_TXT[] = "Falsche Return ID"
    CASE 344
      USER_MSG.MSG_TXT[] = "Abbruch durch User"
      SK[1] = {Sk_Type #Value,Sk_Txt[] "OK"}
    CASE 345
      USER_MSG.MSG_TXT[] = "Reset durchfuehren"
      SK[2] = {Sk_Type #Value,Sk_Txt[] "Reset"}
;	Fehler (Messende)
    CASE 400
  		USER_MSG.MSG_TXT[] = "Erfolgreich"
    CASE 404
  		USER_MSG.MSG_TXT[] = "Timeout: Beim warten auf I_PRC_MEACK"
      $FLAG[F_PRC_TmOut]=TRUE
    CASE 424
      USER_MSG.MSG_TXT[] = "System nicht gestartet"
    CASE 426
  		USER_MSG.MSG_TXT[] = "Timeout: Beim warten auf I_PRC_DaSend"
      $FLAG[F_PRC_TmOut]=TRUE
    CASE 427
  		USER_MSG.MSG_TXT[] = "Timeout: Beim warten auf I_PRC_DaNew"
      $FLAG[F_PRC_TmOut]=TRUE
    CASE 428
  		USER_MSG.MSG_TXT[] = "Timeout: Beim warten auf nicht I_PRC_DaNew"
      $FLAG[F_PRC_TmOut]=TRUE
    CASE 434
  		USER_MSG.MSG_TXT[] = "Falsche PunktFolge"
    CASE 435
  		USER_MSG.MSG_TXT[] = "Anzahl MP zu klein u. falsche PunktFolge"
    CASE 436
  		USER_MSG.MSG_TXT[] = "Ungueltiger PAR_1 bei Messende"
    CASE 437
  		USER_MSG.MSG_TXT[] = "Anzahl MP zu klein"
    CASE 443
      USER_MSG.MSG_TXT[] = "Falsche Return ID"
;	Fehler (Reset)
    CASE 500
  		USER_MSG.MSG_TXT[] = "Erfolgreich"
    CASE 521
  		USER_MSG.MSG_TXT[] = "Timeout: Beim warten auf I_PRC_Reset"
      $FLAG[F_PRC_TmOut]=TRUE
      SK[2] = {Sk_Type #Value,Sk_Txt[] "Wdh."}
    CASE 522
  		USER_MSG.MSG_TXT[] = "Timeout: Beim warten auf nicht I_PRC_Reset"
      $FLAG[F_PRC_TmOut]=TRUE
      SK[2] = {Sk_Type #Value,Sk_Txt[] "Wdh."}
;	Fehler (Sensortausch)
    CASE 600
  		USER_MSG.MSG_TXT[] = "gestartet"
    CASE 601
      USER_MSG.MSG_TXT[] = "Timeout: Beim Sendekanal oeffnen"
      $FLAG[F_PRC_TmOut]=TRUE
    CASE 602
      USER_MSG.MSG_TXT[] = "Timeout: Beim warten auf I_PRC_DaComp"
      $FLAG[F_PRC_TmOut]=TRUE
    CASE 603
      USER_MSG.MSG_TXT[] = "Timeout: Beim warten auf nicht I_PRC_DaComp"
      $FLAG[F_PRC_TmOut]=TRUE
    CASE 604
      USER_MSG.MSG_TXT[] = "Timeout: Beim warten auf I_PRC_MEACK"
      $FLAG[F_PRC_TmOut]=TRUE
    CASE 605
  		USER_MSG.MSG_TXT[] = "Modell oder Routine nicht definiert"
      SK[2] = {Sk_Type #Value,Sk_Txt[] "Wdh."}
      MLD_TYP = #DlgMsg
    CASE 606
  		USER_MSG.MSG_TXT[] = "System in Automatikmodus schalten"
      SK[1] = {Sk_Type #Empty}
      SK[2] = {Sk_Type #Value,Sk_Txt[] "Wdh."}
    CASE 607
  		USER_MSG.MSG_TXT[] = "System bereits gestartet"
      SK[2] = {Sk_Type #Value,Sk_Txt[] "Reset"}
    CASE 608
  		USER_MSG.MSG_TXT[] = "Fehler allgemein"
    CASE 609
  		USER_MSG.MSG_TXT[] = "Fehler nicht spezifiziert"
    CASE 610
  		USER_MSG.MSG_TXT[] = "Sensormontage pruefen"
      SK[1] = {Sk_Type #Value,Sk_Txt[] "Abbr."}
      SK[2] = {Sk_Type #Value,Sk_Txt[] "Wdh."}
    CASE 611
  		USER_MSG.MSG_TXT[] = "System mit anderem Modell gestartet"
    CASE 612
  		USER_MSG.MSG_TXT[] = "System von der SPS gestartet"
    CASE 613
      USER_MSG.MSG_TXT[] = "Fehler allgemein"
    CASE 617
      USER_MSG.MSG_TXT[] = "Timeout: Beim Daten Senden"
      $FLAG[F_PRC_TmOut]=TRUE
    CASE 618
      USER_MSG.MSG_TXT[] = "Daten nicht gespiegelt"
    CASE 623
      USER_MSG.MSG_TXT[] = "Positionsnummer ungueltig"
    CASE 624
      USER_MSG.MSG_TXT[] = "System nicht gestartet"
    CASE 625
      USER_MSG.MSG_TXT[] = "Falsche Punktreihenfolge"
    CASE 626
  		USER_MSG.MSG_TXT[] = "Timeout: Beim warten auf I_PRC_DaSend"
      $FLAG[F_PRC_TmOut]=TRUE
    CASE 627
  		USER_MSG.MSG_TXT[] = "Timeout: Beim warten auf I_PRC_DaNew"
      $FLAG[F_PRC_TmOut]=TRUE
    CASE 628
      USER_MSG.MSG_TXT[] = "Timeout: Beim warten auf nicht I_PRC_DaNew"
      $FLAG[F_PRC_TmOut]=TRUE
    CASE 629
      USER_MSG.MSG_TXT[] = "Routinennummer ist 0"
    CASE 630
  		USER_MSG.MSG_TXT[] = "Bitte System in den Kalibriermodus schalten"
    CASE 631
      SWRITE(USER_MSG.MSG_TXT[],STATE,OFFSET,"Falscher Status vom System: %d",nTmp)
      SK[2] = {Sk_Type #Value,Sk_Txt[] "Wdh."}
    CASE 632
  		USER_MSG.MSG_TXT[] = "System nicht im Kalibriermodus"
      SK[1] = {Sk_Type #Empty}
      SK[2] = {Sk_Type #Value,Sk_Txt[] "Wdh."}
    CASE 633
  		USER_MSG.MSG_TXT[] = "Pruefen Erfolgreich"
      SK[1] = {Sk_Type #Value,Sk_Txt[] "Weiter"}
    CASE 634
  		USER_MSG.MSG_TXT[] = "Falsche PunktFolge"
    CASE 635
  		USER_MSG.MSG_TXT[] = "Anzahl Messpunkte zu klein u. falsche PunktFolge"
    CASE 636
  		USER_MSG.MSG_TXT[] = "Ungueltiger PAR_1 bei Messende"
    CASE 637
  		USER_MSG.MSG_TXT[] = "Anzahl Messpunkte zu klein"
    CASE 638
  		USER_MSG.MSG_TXT[] = "Kalibrierung erforderlich"
    CASE 639
  		USER_MSG.MSG_TXT[] = "Nur im SingleStep-Betrieb moeglich"
      SK[1] = {Sk_Type #Value,Sk_Txt[] "OK"}
   CASE 640
      swrite(USER_MSG.MSG_TXT[],STATE,OFFSET,"UP Mod: %d/Rout: %d nicht definiert; DAT bearbeiten",nTmp,nPar)
    CASE 641
      swrite(USER_MSG.MSG_TXT[],STATE,OFFSET,"UP Mod: %d/Rout: %d ist 0; DAT bearbeiten",nTmp,nPar)
    CASE 643
      USER_MSG.MSG_TXT[] = "Falsche Return ID"
    CASE 644
      USER_MSG.MSG_TXT[] = "Abbruch durch User"
      SK[1] = {Sk_Type #Value,Sk_Txt[] "OK"}
    CASE 650
  		USER_MSG.MSG_TXT[] = "Bitte System in den Toolfindermodus schalten"
    CASE 652
  		USER_MSG.MSG_TXT[] = "System nicht im Toolfindermodus"
      SK[1] = {Sk_Type #Empty}
      SK[2] = {Sk_Type #Value,Sk_Txt[] "Wdh."}
    CASE 653
  		USER_MSG.MSG_TXT[] = "Toolfinder berechnen und anwenden!"
      SK[1] = {Sk_Type #Value,Sk_Txt[] "OK"}
    CASE 698
  		USER_MSG.MSG_TXT[] = "Sensortausch erfolgreich durchgefuehrt"
      SK[1] = {Sk_Type #Value,Sk_Txt[] "OK"}
    CASE 699
  		USER_MSG.MSG_TXT[] = "Kalibrierung pruefen"
      SK[1] = {Sk_Type #Value,Sk_Txt[] "OK"}
;	Fehler (Robotertausch)
    CASE 700
  		USER_MSG.MSG_TXT[] = "Abgeschlossen"
    CASE 701
  		USER_MSG.MSG_TXT[] = "Timeout: Beim Sendekanal oeffnen"
      $FLAG[F_PRC_TmOut]=TRUE
    CASE 702
      USER_MSG.MSG_TXT[] = "Timeout: Beim warten auf I_PRC_DaComp"
      $FLAG[F_PRC_TmOut]=TRUE
    CASE 703
      USER_MSG.MSG_TXT[] = "Timeout: Beim warten auf nicht I_PRC_DaComp"
      $FLAG[F_PRC_TmOut]=TRUE
    CASE 704
      USER_MSG.MSG_TXT[] = "Timeout: Beim warten auf I_PRC_MEACK"
      $FLAG[F_PRC_TmOut]=TRUE
    CASE 705
  		USER_MSG.MSG_TXT[] = "Modell oder Routine nicht definiert"
      SK[2] = {Sk_Type #Value,Sk_Txt[] "Wdh."}
      MLD_TYP = #DlgMsg
    CASE 706
      USER_MSG.MSG_TXT[] = "System in Automatikmodus schalten"
      SK[1] = {Sk_Type #Empty}
      SK[2] = {Sk_Type #Value,Sk_Txt[] "Wdh."}
    CASE 707
  		USER_MSG.MSG_TXT[] = "System bereits gestartet"
      SK[2] = {Sk_Type #Value,Sk_Txt[] "Reset"}
    CASE 708
  		USER_MSG.MSG_TXT[] = "Fehler allgemein"
    CASE 709
  		USER_MSG.MSG_TXT[] = "Fehler nicht spezifiziert"
    CASE 710
  		USER_MSG.MSG_TXT[] = "Robotermontage pruefen"
      SK[1] = {Sk_Type #Value,Sk_Txt[] "Abbr."}
      SK[2] = {Sk_Type #Value,Sk_Txt[] "Wdh."}
    CASE 711
  		USER_MSG.MSG_TXT[] = "System mit anderem Modell gestartet"
    CASE 712
  		USER_MSG.MSG_TXT[] = "System von der SPS gestartet"
    CASE 713
      USER_MSG.MSG_TXT[] = "Fehler allgemein"
    CASE 714
  		USER_MSG.MSG_TXT[] = "Keine Korrekturwerte vorhanden"
      $FLAG[F_PRC_TmOut]=TRUE
    CASE 718
    CASE 723
      USER_MSG.MSG_TXT[] = "Positionsnummer ungueltig"
    CASE 724
      USER_MSG.MSG_TXT[] = "System nicht gestartet"
    CASE 725
      USER_MSG.MSG_TXT[] = "Falsche Punktreihenfolge"
    CASE 726
  		USER_MSG.MSG_TXT[] = "Timeout: Beim warten auf I_PRC_DaSend"
      $FLAG[F_PRC_TmOut]=TRUE
    CASE 727
  		USER_MSG.MSG_TXT[] = "Timeout: Beim warten auf I_PRC_DaNew"
      $FLAG[F_PRC_TmOut]=TRUE
    CASE 728
      USER_MSG.MSG_TXT[] = "Timeout: Beim warten auf nicht I_PRC_DaNew"
      $FLAG[F_PRC_TmOut]=TRUE
    CASE 729
      USER_MSG.MSG_TXT[] = "Routinennummer ist 0"
    CASE 730
  		USER_MSG.MSG_TXT[] = "Bitte System in den Automatik-Modus schalten"
    CASE 731
      SWRITE(USER_MSG.MSG_TXT[],STATE,OFFSET,"Falscher Status vom System: %d",nTmp)
      SK[2] = {Sk_Type #Value,Sk_Txt[] "Wdh."}
    CASE 732
  		USER_MSG.MSG_TXT[] = "System nicht im Automatik-Modus"
      SK[1] = {Sk_Type #Empty}
      SK[2] = {Sk_Type #Value,Sk_Txt[] "Wdh."}
    CASE 733
  		USER_MSG.MSG_TXT[] = "Pruefen Erfolgreich"
      SK[1] = {Sk_Type #Value,Sk_Txt[] "Weiter"}
    CASE 734
      USER_MSG.MSG_TXT[] = "Falsche PunktFolge"
    CASE 735
  		USER_MSG.MSG_TXT[] = "Anzahl Messpunkte zu klein u. falsche PunktFolge"
    CASE 736
  		USER_MSG.MSG_TXT[] = "Ungueltiger PAR_1 bei Messende"
    CASE 737
  		USER_MSG.MSG_TXT[] = "Anzahl Messpunkte zu klein"
    CASE 739
  		USER_MSG.MSG_TXT[] = "Nur im SingleStep-Betrieb moeglich"
      SK[1] = {Sk_Type #Value,Sk_Txt[] "OK"}
    CASE 740
      swrite(USER_MSG.MSG_TXT[],STATE,OFFSET,"UP Mod: %d/Rout: %d nicht definiert; DAT bearbeiten",nTmp,nPar)
    CASE 741
      swrite(USER_MSG.MSG_TXT[],STATE,OFFSET,"UP Mod: %d/Rout: %d ist 0; DAT bearbeiten",nTmp,nPar)
    CASE 743
      USER_MSG.MSG_TXT[] = "Falsche Return ID"
    CASE 744
      USER_MSG.MSG_TXT[] = "Abbruch durch User"
      SK[1] = {Sk_Type #Value,Sk_Txt[] "OK"}
    CASE 795
  		USER_MSG.MSG_TXT[] = "Rob.Pos ungueltig schalten"
    CASE 796
  		USER_MSG.MSG_TXT[] = "Toolfinder berechnen und anwenden!"
      SK[1] = {Sk_Type #Value,Sk_Txt[] "OK"}
    CASE 797
  		USER_MSG.MSG_TXT[] = "Korrektur notwendig, Basekorr. wird ausgefuehrt"
      SK[1] = {Sk_Type #Value,Sk_Txt[] "OK"}
    CASE 798
  		USER_MSG.MSG_TXT[] = "Robotertausch erfolgreich durchgefuehrt"
      SK[1] = {Sk_Type #Value,Sk_Txt[] "OK"}
    CASE 799
  		USER_MSG.MSG_TXT[] = "Kalibrierung pruefen"
      SK[1] = {Sk_Type #Value,Sk_Txt[] "OK"}
;	Fehler (Hole UP-Nr)
    CASE 800
  		USER_MSG.MSG_TXT[] = "Erfolgreich"
    CASE 801
      USER_MSG.MSG_TXT[] = "Timeout: Beim Sendekanal oeffnen"
      $FLAG[F_PRC_TmOut]=TRUE
      SK[1] = {Sk_Type #Value,Sk_Txt[] "OK"}
      MLD_TYP = #DlgMsg
    CASE 802
      USER_MSG.MSG_TXT[] = "Timeout: Beim warten auf IN_DataComplete"
      $FLAG[F_PRC_TmOut]=TRUE
      SK[1] = {Sk_Type #Value,Sk_Txt[] "OK"}
      MLD_TYP = #DlgMsg
    CASE 803
      USER_MSG.MSG_TXT[] = "Timeout: Beim warten auf nicht IN_DataComplete"
      $FLAG[F_PRC_TmOut]=TRUE
      SK[1] = {Sk_Type #Value,Sk_Txt[] "OK"}
      MLD_TYP = #DlgMsg
    CASE 804
      USER_MSG.MSG_TXT[] = "Timeout: Beim warten auf I_PRC_MEACK"
      $FLAG[F_PRC_TmOut]=TRUE
      SK[1] = {Sk_Type #Value,Sk_Txt[] "OK"}
      MLD_TYP = #DlgMsg
    CASE 805
      USER_MSG.MSG_TXT[] = "Modell od. Routine nicht definiert"
      SK[1] = {Sk_Type #Value,Sk_Txt[] "OK"}
      MLD_TYP = #DlgMsg
    CASE 806
      USER_MSG.MSG_TXT[] = "System im Offline/Programmier-Modus"
      SK[1] = {Sk_Type #Value,Sk_Txt[] "OK"}
      SK[3] = {Sk_Type #Value,Sk_Txt[] "Wdh."}
      MLD_TYP = #DlgMsg
    CASE 807
      USER_MSG.MSG_TXT[] = "System von SPS nicht gestartet"
      SK[3] = {Sk_Type #Value,Sk_Txt[] "Wdh."}
      MLD_TYP = #DlgMsg
    CASE 808
      USER_MSG.MSG_TXT[] = "Fehler allgemein"
      SK[1] = {Sk_Type #Value,Sk_Txt[] "OK"}
      SK[2] = {Sk_Type #Value,Sk_Txt[] "Reset"}
      MLD_TYP = #DlgMsg
    CASE 809
      USER_MSG.MSG_TXT[] = "System Fehler nicht spezifiziert"
      SK[1] = {Sk_Type #Value,Sk_Txt[] "OK"}
      SK[2] = {Sk_Type #Value,Sk_Txt[] "Reset"}
      MLD_TYP = #DlgMsg
    CASE 811
      USER_MSG.MSG_TXT[] = "System mit anderem Modell bereits gestartet"
      SK[1] = {Sk_Type #Value,Sk_Txt[] "OK"}
      SK[2] = {Sk_Type #Value,Sk_Txt[] "Reset"}
      MLD_TYP = #DlgMsg
    CASE 817
      USER_MSG.MSG_TXT[] = "Timeout: Beim Daten senden"
      $FLAG[F_PRC_TmOut]=TRUE
      SK[1] = {Sk_Type #Value,Sk_Txt[] "OK"}
      MLD_TYP = #DlgMsg
    CASE 818
      USER_MSG.MSG_TXT[] = "Daten nicht gespiegelt"
      SK[1] = {Sk_Type #Value,Sk_Txt[] "OK"}
      MLD_TYP = #DlgMsg
    CASE 827
      USER_MSG.MSG_TXT[] = "Timeout: Beim warten auf I_PRC_DaNew"
      SK[1] = {Sk_Type #Value,Sk_Txt[] "OK"}
      MLD_TYP = #DlgMsg
    CASE 828
      USER_MSG.MSG_TXT[] = "Timeout: Beim warten auf nicht I_PRC_DaNew"
      $FLAG[F_PRC_TmOut]=TRUE
      SK[1] = {Sk_Type #Value,Sk_Txt[] "OK"}
      MLD_TYP = #DlgMsg
    CASE 829
      USER_MSG.MSG_TXT[] = "Routinennummer ist 0"
      SK[1] = {Sk_Type #Value,Sk_Txt[] "OK"}
      MLD_TYP = #DlgMsg
    CASE 840
      swrite(USER_MSG.MSG_TXT[],STATE,OFFSET,"UP Mod: %d/Rout: %d Aufruf nicht definiert; In .DAT einfuegen",nTmp,nPar)
      SK[1] = {Sk_Type #Value,Sk_Txt[] "OK"}
      MLD_TYP = #DlgMsg
    CASE 841
      swrite(USER_MSG.MSG_TXT[],STATE,OFFSET,"UP Mod: %d/Rout: %d Antwort nicht definiert; In .DAT einfuegen",nTmp,nPar)
      SK[1] = {Sk_Type #Value,Sk_Txt[] "OK"}
      MLD_TYP = #DlgMsg
    CASE 843
      USER_MSG.MSG_TXT[] = "Falsche Return ID"
      SK[1] = {Sk_Type #Value,Sk_Txt[] "OK"}
      MLD_TYP = #DlgMsg
	CASE 850
      USER_MSG.MSG_TXT[] = "Kompensation OK"
    CASE 851
      USER_MSG.MSG_TXT[] = "Kompensation erford. (Voll)"
    CASE 852
      USER_MSG.MSG_TXT[] = "Kompensation erford. (Split)"
    CASE 853
      USER_MSG.MSG_TXT[] = "Kompensation deaktiviert (SPS)"
    CASE 854
      USER_MSG.MSG_TXT[] = "Modell/UP ungueltig"
    CASE 860
      USER_MSG.MSG_TXT[] = "Startprozedur laeuft (Status)"
    CASE 861
      USER_MSG.MSG_TXT[] = "Startprozedur laeuft (Programm)"
    CASE 870
      USER_MSG.MSG_TXT[] = "Fehler in der Startprozedur"
      SK[1] = {Sk_Type #Value,Sk_Txt[] "OK"}
      MLD_TYP = #DlgMsg
    CASE 871
      USER_MSG.MSG_TXT[] = "Kompensation NOK (Konfiguration)"
      SK[1] = {Sk_Type #Value,Sk_Txt[] "OK"}
      MLD_TYP = #DlgMsg
    CASE 872
      swrite(USER_MSG.MSG_TXT[],STATE,OFFSET,"Modell-Freigabe: %d ungueltig",nTmp)
      SK[1] = {Sk_Type #Value,Sk_Txt[] "OK"}
      MLD_TYP = #DlgMsg
    CASE 873
      swrite(USER_MSG.MSG_TXT[],STATE,OFFSET,"Modell-Freigabe: %d = Aus fuer das Modell",nTmp)
      SK[1] = {Sk_Type #Value,Sk_Txt[] "OK"}
      MLD_TYP = #DlgMsg
;	Fehler (Ungueltige Parameter)
    CASE 900
  		USER_MSG.MSG_TXT[] = "Gueltig"
    CASE 901
      SWRITE(USER_MSG.MSG_TXT[],STATE,OFFSET,"Modus %d ungueltig (1001-1003)",nTmp)
      MLD_TYP = #DlgMsg
    CASE 902
      SWRITE(USER_MSG.MSG_TXT[],STATE,OFFSET,"Funktion %d im Modus %d ungueltig",nTmp,nPar)
      MLD_TYP = #DlgMsg
    CASE 903
      SWRITE(USER_MSG.MSG_TXT[],STATE,OFFSET,"Modell %d ungueltig (1 <> 65535)",nTmp)
      MLD_TYP = #DlgMsg
    CASE 904
      SWRITE(USER_MSG.MSG_TXT[],STATE,OFFSET,"Parameter 2 %d ungueltig (0 <> 65535)",nTmp)
      MLD_TYP = #DlgMsg
    CASE 905
      SWRITE(USER_MSG.MSG_TXT[],STATE,OFFSET,"Parameter 3 %d ungueltig (0 <> 256)",nTmp)
      MLD_TYP = #DlgMsg
    CASE 906
      SWRITE(USER_MSG.MSG_TXT[],STATE,OFFSET,"Parameter 4 %d ungueltig (-180 <> 65535)",nTmp)
      MLD_TYP = #DlgMsg
    CASE 907
      SWRITE(USER_MSG.MSG_TXT[],STATE,OFFSET,"Parameter 5 %d ungueltig (-180 <> 255)",nTmp)
      MLD_TYP = #DlgMsg
	CASE 908
      SWRITE(USER_MSG.MSG_TXT[],STATE,OFFSET,"Parameter 6 %d ungueltig (-180 <> 255)",nTmp)
      MLD_TYP = #DlgMsg
    CASE 910
      SWRITE(USER_MSG.MSG_TXT[],STATE,OFFSET,"Modus %d mit Funktion %d ungueltig",nTmp,nPar)
      MLD_TYP = #DlgMsg
    CASE 911
      SWRITE(USER_MSG.MSG_TXT[],STATE,OFFSET,"Kommando %d ungueltig",nTmp)
      MLD_TYP = #DlgMsg
;	Fehler (Hole Korrektur)
    CASE 1000
  		USER_MSG.MSG_TXT[] = "Erfolgreich"
    CASE 1001
      USER_MSG.MSG_TXT[] = "Timeout: Beim Sendekanal oeffnen"
      $FLAG[F_PRC_TmOut]=TRUE
    CASE 1002
      USER_MSG.MSG_TXT[] = "Timeout: Beim warten auf I_PRC_DaComp"
      $FLAG[F_PRC_TmOut]=TRUE
    CASE 1003
      USER_MSG.MSG_TXT[] = "Timeout: Beim warten auf nicht I_PRC_DaComp"
      $FLAG[F_PRC_TmOut]=TRUE
    CASE 1004
      USER_MSG.MSG_TXT[] = "Timeout: Beim warten auf I_PRC_MEACK"
      $FLAG[F_PRC_TmOut]=TRUE
    CASE 1005
  		USER_MSG.MSG_TXT[] = "Modell oder Routine nicht definiert"
      SK[2] = {Sk_Type #Value,Sk_Txt[] "Reset"}
    CASE 1006
  		USER_MSG.MSG_TXT[] = "System im Offline/Programmier-Modus"
      SK[3] = {Sk_Type #Value,Sk_Txt[] "Wdh."}
    CASE 1007
  		USER_MSG.MSG_TXT[] = "System bereits gestartet"
      SK[2] = {Sk_Type #Value,Sk_Txt[] "Reset"}
    CASE 1008
  		USER_MSG.MSG_TXT[] = "Fehler allgemein"
      SK[2] = {Sk_Type #Value,Sk_Txt[] "Reset"}
    CASE 1009
  		USER_MSG.MSG_TXT[] = "Fehler nicht spezifiziert"
      SK[2] = {Sk_Type #Value,Sk_Txt[] "Reset"}
    CASE 1011
  		USER_MSG.MSG_TXT[] = "System mit anderem Modell gestartet"
      SK[2] = {Sk_Type #Value,Sk_Txt[] "Reset"}
    CASE 1012
  		USER_MSG.MSG_TXT[] = "System von der SPS gestartet"
      SK[2] = {Sk_Type #Value,Sk_Txt[] "Reset"}
    CASE 1017
      USER_MSG.MSG_TXT[] = "Timeout: Beim Daten Senden"
      $FLAG[F_PRC_TmOut]=TRUE
    CASE 1018
      USER_MSG.MSG_TXT[] = "Fehler: Beim Daten spiegeln"
    CASE 1019
      USER_MSG.MSG_TXT[] = "Werte ueberschreiten VF_PRC_Min"
    CASE 1020
      USER_MSG.MSG_TXT[] = "Werte ueberschreiten VF_PRC_Max"
    CASE 1027
      USER_MSG.MSG_TXT[] = "Timeout: Beim warten auf I_PRC_DaNew"
      $FLAG[F_PRC_TmOut]=TRUE
    CASE 1028
      USER_MSG.MSG_TXT[] = "Timeout: Beim warten auf nicht I_PRC_DaNew"
      $FLAG[F_PRC_TmOut]=TRUE
    CASE 1038
      USER_MSG.MSG_TXT[] = "Falsche Return Korrekturnummer"
    CASE 1042
      USER_MSG.MSG_TXT[] = "keine Korrekturwerte vorhanden"
    CASE 1043
      USER_MSG.MSG_TXT[] = "Falsche Return ID"
    CASE 1046
      USER_MSG.MSG_TXT[] = "Korrekturwerte nicht umgesetzt"
;	Fehler (Alarme)
    CASE 1100
  		USER_MSG.MSG_TXT[] = "Erfolgreich"
    CASE 1101
      USER_MSG.MSG_TXT[] = "Trend"
      SK[1] = {Sk_Type #Value,Sk_Txt[] "OK"}
    CASE 1102
      USER_MSG.MSG_TXT[] = "Toleranz"
      SK[1] = {Sk_Type #Value,Sk_Txt[] "OK"}
    CASE 1103
      USER_MSG.MSG_TXT[] = "Toleranz, Trend"
      SK[1] = {Sk_Type #Value,Sk_Txt[] "OK"}
    CASE 1104
      USER_MSG.MSG_TXT[] = "Ausschuss"
      SK[1] = {Sk_Type #Value,Sk_Txt[] "OK"}
    CASE 1105
      USER_MSG.MSG_TXT[] = "Ausschuss, Trend"
      SK[1] = {Sk_Type #Value,Sk_Txt[] "OK"}
    CASE 1106
      USER_MSG.MSG_TXT[] = "Ausschuss, Toleranz"
      SK[1] = {Sk_Type #Value,Sk_Txt[] "OK"}
    CASE 1107
      USER_MSG.MSG_TXT[] = "Ausschuss, Toleranz, Trend"
      SK[1] = {Sk_Type #Value,Sk_Txt[] "OK"}
    CASE 1108
      USER_MSG.MSG_TXT[] = "Error"
      SK[1] = {Sk_Type #Value,Sk_Txt[] "OK"}
    CASE 1151
      USER_MSG.MSG_TXT[] = "Roboter.1 Error"
      SK[1] = {Sk_Type #Value,Sk_Txt[] "OK"}
    CASE 1152
      USER_MSG.MSG_TXT[] = "Roboter.1 Toleranz"
      SK[1] = {Sk_Type #Value,Sk_Txt[] "OK"}
    CASE 1153
      USER_MSG.MSG_TXT[] = "Roboter.1 VF Error"
      SK[1] = {Sk_Type #Value,Sk_Txt[] "OK"}
    CASE 1154
      USER_MSG.MSG_TXT[] = "Roboter.1 VF Toleranz"
      SK[1] = {Sk_Type #Value,Sk_Txt[] "OK"}
    CASE 1155
      USER_MSG.MSG_TXT[] = "Roboter.2 Error"
      SK[1] = {Sk_Type #Value,Sk_Txt[] "OK"}
    CASE 1156
      USER_MSG.MSG_TXT[] = "Roboter.2 Toleranz"
      SK[1] = {Sk_Type #Value,Sk_Txt[] "OK"}
    CASE 1157
      USER_MSG.MSG_TXT[] = "Roboter.2 VF Error"
      SK[1] = {Sk_Type #Value,Sk_Txt[] "OK"}
    CASE 1158
      USER_MSG.MSG_TXT[] = "Roboter.2 VF Toleranz"
      SK[1] = {Sk_Type #Value,Sk_Txt[] "OK"}
    CASE 1159
      USER_MSG.MSG_TXT[] = "Roboter.1 mehrere Fehler"
      SK[1] = {Sk_Type #Value,Sk_Txt[] "OK"}
    CASE 1160
      USER_MSG.MSG_TXT[] = "Roboter.2 mehrere Fehler"
      SK[1] = {Sk_Type #Value,Sk_Txt[] "OK"}
;  Init
	CASE 1200
      swrite(USER_MSG.MSG_TXT[],STATE,OFFSET,"Falsches Subsystem: %d",nPar)
      SK[1] = {Sk_Type #Value,Sk_Txt[] "OK"}
      MLD_TYP = #DlgMsg
	CASE 1201
      swrite(USER_MSG.MSG_TXT[],STATE,OFFSET,"Falsches Conveyor-Tech: %d",nTmp)
      SK[1] = {Sk_Type #Value,Sk_Txt[] "OK"}
      MLD_TYP = #DlgMsg
	CASE 1202
      swrite(USER_MSG.MSG_TXT[],STATE,OFFSET,"Falsches Frame: %d",nTmp)
      SK[1] = {Sk_Type #Value,Sk_Txt[] "OK"}
      MLD_TYP = #DlgMsg
	CASE 1210
      swrite(USER_MSG.MSG_TXT[],STATE,OFFSET,"Falsches Modell[%d]: %d",nTmp,nPar)
      SK[1] = {Sk_Type #Value,Sk_Txt[] "OK"}
      MLD_TYP = #DlgMsg
	CASE 1215
      swrite(USER_MSG.MSG_TXT[],STATE,OFFSET,"Falsches Translation/Rotation [MIN]: %d",nTmp)
      SK[1] = {Sk_Type #Value,Sk_Txt[] "OK"}
      MLD_TYP = #DlgMsg
	CASE 1216
      swrite(USER_MSG.MSG_TXT[],STATE,OFFSET,"Falsches Translation/Rotation [MAX]: %d",nTmp)
      SK[1] = {Sk_Type #Value,Sk_Txt[] "OK"}
      MLD_TYP = #DlgMsg
	CASE 1217
      swrite(USER_MSG.MSG_TXT[],STATE,OFFSET,"Falsches Min/Max: %d",nTmp)
      SK[1] = {Sk_Type #Value,Sk_Txt[] "OK"}
      MLD_TYP = #DlgMsg
;  Version
    CASE 9000
      swrite(USER_MSG.MSG_TXT[],STATE,OFFSET,"Major-Nr: %d Minor-Nr: %d Revisions-Nr: %d",N_PRC_VerMaj,N_PRC_VerMin,N_PRC_VerRev)
      SK[1] = {Sk_Type #Value,Sk_Txt[] "OK"}
      MLD_TYP = #DlgMsg
;	Fehler: (Unbekannt)
    DEFAULT
      swrite(USER_MSG.MSG_TXT[],STATE,OFFSET,"Unbekannter Fehler %d",MSG_NR)
      SK[1] = {Sk_Type #Value,Sk_Txt[] "OK"}
  ENDSWITCH
;
  ;ENDFOLD (Meldungs-Nr)
;
  IF MSG_NR > 0 THEN
    USER_MSG.Nr = MSG_NR
  ENDIF
  OFFSET      = 0
  SWRITE(USER_MSG.MSG_TXT[],STATE,OFFSET,"%s %s",sMeldFunction[],USER_MSG.MSG_TXT[])
  IF (($mode_op == #T1) OR ($mode_op == #T2)) THEN
    MLD_TYP = #DlgMsg
  ENDIF
  nDlgAnswer = 1
  SWITCH MLD_TYP
    CASE #DlgMsg
      nDlgHandle = Set_KrlDlg(USER_MSG,Par[],SK[],Opt)
      IF (nDlgHandle > 0) Then
        While (Exists_KrlDlg(nDlgHandle, nDlgAnswer))         ;Warten bis der Dialog beantwortet wird
          Wait Sec 0.1
        ENDWHILE
        SWITCH nDlgAnswer
          CASE 1
            ;HALT ;Softkey 1 was hit
          CASE 2
            ;HALT ;Softkey 2 was hit
          CASE 3
            ;HALT ;Softkey 3 was hit
          DEFAULT
            ;HALT ;Wrong softkey was hit
        ENDSWITCH
      ENDIF
    CASE #StatMsg
      nDlgHandle = Set_KrlMsg (#State, USER_MSG, Par[], OPT)   ; Ausgabe Statusmeldung
    CASE #QuitMsg
      nDlgHandle = Set_KrlMsg (#Quit, USER_MSG, Par[], OPT)    ; Ausgabe Quittierungsmeldung
      IF (nDlgHandle > 0) Then
        While ( Exists_KrlMsg(nDlgHandle))                     ;Warten bis der Anwender quittiert
          Wait Sec 0.1
        ENDWHILE
      ENDIF
    CASE #NotifyMsg
      nDlgHandle = Set_KrlMsg (#Notify, USER_MSG, Par[], Opt)  ; Ausgabe Hinweismeldung
    CASE #WaitMsg
      nDlgHandle = Set_KrlMsg (#Waiting, USER_MSG, Par[], Opt) ; Ausgabe Hinweismeldung
    DEFAULT
      USER_MSG.MSG_TXT[] = "MSG_Typ falsch"
      nDlgHandle = Set_KrlMsg (#Quit, USER_MSG, Par[], OPT)    ; Ausgabe Quittierungsmeldung
      IF (nDlgHandle > 0) Then
        While (Exists_KrlMsg(nDlgHandle))                      ;Warten bis der Anwender quittiert
          Wait Sec 0.1
        ENDWHILE
      ENDIF
  ENDSWITCH
  RETURN(nDlgAnswer)
ENDFCT
;
;ENDFOLD (Fehlermeldungen)
;
;endfold

